C01810=1204.723,228.544,-60.567,-177.311,6.595,148.417
C01811=1204.727,228.295,-60.541,-177.313,6.593,148.418
C01812=1204.732,228.047,-60.516,-177.316,6.591,148.418
C01813=1204.736,227.798,-60.490,-177.318,6.589,148.418
C01814=1204.740,227.549,-60.465,-177.321,6.587,148.418
C01815=1204.745,227.300,-60.440,-177.324,6.586,148.419
C01816=1204.749,227.052,-60.414,-177.326,6.584,148.419
C01817=1204.755,226.803,-60.389,-177.329,6.581,148.419
C01818=1204.759,226.554,-60.364,-177.332,6.579,148.420
C01819=1204.762,226.306,-60.338,-177.334,6.577,148.420
C01820=1204.767,226.057,-60.314,-177.337,6.575,148.420
C01821=1204.772,225.808,-60.288,-177.339,6.573,148.420
C01822=1204.776,225.560,-60.263,-177.342,6.571,148.421
C01823=1204.781,225.311,-60.238,-177.344,6.569,148.421
C01824=1204.786,225.063,-60.212,-177.347,6.567,148.421
C01825=1204.790,224.814,-60.187,-177.350,6.565,148.421
C01826=1204.794,224.565,-60.162,-177.352,6.563,148.422
C01827=1204.799,224.316,-60.137,-177.355,6.561,148.422
C01828=1204.804,224.068,-60.112,-177.358,6.559,148.422
C01829=1204.808,223.819,-60.086,-177.360,6.557,148.423
C01830=1204.813,223.570,-60.062,-177.362,6.555,148.423
C01831=1204.817,223.321,-60.036,-177.365,6.553,148.423
C01832=1204.821,223.072,-60.011,-177.368,6.551,148.423
C01833=1204.826,222.824,-59.986,-177.371,6.549,148.424
C01834=1204.830,222.575,-59.961,-177.373,6.547,148.424
C01835=1204.835,222.327,-59.936,-177.376,6.545,148.424
C01836=1204.840,222.078,-59.912,-177.378,6.543,148.424
C01837=1204.844,221.829,-59.886,-177.381,6.541,148.425
C01838=1204.849,221.581,-59.861,-177.384,6.539,148.425
C01839=1204.853,221.332,-59.835,-177.386,6.537,148.425
C01840=1204.858,221.084,-59.811,-177.388,6.535,148.426
C01841=1204.862,220.834,-59.786,-177.391,6.533,148.426
C01842=1204.867,220.586,-59.761,-177.394,6.531,148.426
C01843=1204.872,220.337,-59.736,-177.397,6.529,148.427
C01844=1204.876,220.089,-59.711,-177.399,6.527,148.427
C01845=1204.880,219.839,-59.686,-177.402,6.525,148.427
C01846=1204.885,219.591,-59.661,-177.404,6.523,148.427
C01847=1204.889,219.342,-59.636,-177.407,6.521,148.428
C01848=1204.894,219.093,-59.612,-177.410,6.519,148.428
C01849=1204.899,218.845,-59.587,-177.412,6.517,148.428
C01850=1204.903,218.596,-59.562,-177.414,6.515,148.428
C01851=1204.908,218.347,-59.537,-177.417,6.514,148.429
C01852=1204.912,218.098,-59.512,-177.420,6.511,148.429
C01853=1204.916,217.850,-59.487,-177.423,6.509,148.429
C01854=1204.921,217.601,-59.462,-177.425,6.507,148.430
C01855=1204.925,217.352,-59.438,-177.428,6.505,148.430
C01856=1204.930,217.104,-59.413,-177.430,6.503,148.430
C01857=1204.935,216.855,-59.388,-177.433,6.501,148.430
C01858=1204.939,216.606,-59.364,-177.436,6.500,148.431
C01859=1204.944,216.357,-59.339,-177.438,6.498,148.431
C01860=1204.948,216.109,-59.314,-177.441,6.496,148.431
C01861=1204.953,215.860,-59.290,-177.443,6.494,148.432
C01862=1204.957,215.611,-59.264,-177.446,6.492,148.432
C01863=1204.962,215.363,-59.240,-177.449,6.489,148.432
C01864=1204.967,215.114,-59.215,-177.451,6.487,148.433
C01865=1204.971,214.865,-59.191,-177.454,6.486,148.433
C01866=1204.976,214.616,-59.166,-177.457,6.484,148.433
C01867=1204.980,214.368,-59.142,-177.459,6.482,148.433
C01868=1204.985,214.118,-59.117,-177.462,6.480,148.434
C01869=1204.989,213.870,-59.093,-177.464,6.478,148.434
C01870=1204.994,213.622,-59.068,-177.467,6.476,148.434
C01871=1204.998,213.373,-59.043,-177.469,6.474,148.435
C01872=1205.003,213.124,-59.019,-177.472,6.472,148.435
C01873=1205.007,212.876,-58.994,-177.475,6.471,148.435
C01874=1205.012,212.626,-58.969,-177.477,6.468,148.435
C01875=1205.016,212.378,-58.945,-177.480,6.467,148.436
C01876=1205.021,212.129,-58.921,-177.482,6.465,148.436
C01877=1205.025,211.880,-58.896,-177.485,6.463,148.436
C01878=1205.030,211.631,-58.872,-177.488,6.460,148.437
C01879=1205.035,211.361,-58.845,-177.491,6.458,148.437
C01880=1205.040,211.090,-58.819,-177.493,6.457,148.437
C01881=1205.045,210.820,-58.792,-177.496,6.455,148.438
C01882=1205.050,210.549,-58.766,-177.499,6.452,148.438
C01883=1205.054,210.301,-58.742,-177.502,6.450,148.438
C01884=1205.059,210.052,-58.717,-177.504,6.448,148.439
C01885=1205.063,209.803,-58.692,-177.507,6.447,148.439
C01886=1205.067,209.555,-58.668,-177.510,6.445,148.439
C01887=1205.073,209.305,-58.644,-177.512,6.443,148.440
C01888=1205.077,209.057,-58.620,-177.515,6.441,148.440
C01889=1205.082,208.808,-58.595,-177.517,6.439,148.440
C01890=1205.086,208.559,-58.571,-177.520,6.437,148.441
C01891=1205.091,208.311,-58.547,-177.523,6.435,148.441
C01892=1205.096,208.062,-58.523,-177.525,6.433,148.441
C01893=1205.100,207.813,-58.498,-177.528,6.432,148.442
C01894=1205.104,207.564,-58.475,-177.530,6.430,148.442
C01895=1205.109,207.315,-58.450,-177.533,6.428,148.442
C01896=1205.114,207.067,-58.426,-177.536,6.426,148.443
C01897=1205.118,206.818,-58.402,-177.538,6.424,148.443
C01898=1205.123,206.569,-58.377,-177.541,6.422,148.443
C01899=1205.127,206.320,-58.354,-177.543,6.420,148.443
C01900=1205.132,206.071,-58.329,-177.546,6.418,148.444
C01901=1205.136,205.823,-58.305,-177.549,6.417,148.444
C01902=1205.142,205.574,-58.281,-177.551,6.415,148.444
C01903=1205.146,205.325,-58.257,-177.554,6.413,148.445
C01904=1205.150,205.076,-58.233,-177.556,6.411,148.445
C01905=1205.154,204.828,-58.209,-177.559,6.409,148.445
C01906=1205.160,204.578,-58.185,-177.562,6.408,148.446
C01907=1205.164,204.330,-58.161,-177.564,6.406,148.446
C01908=1205.168,204.082,-58.137,-177.567,6.404,148.446
C01909=1205.173,203.833,-58.113,-177.569,6.402,148.447
C01910=1205.178,203.583,-58.088,-177.572,6.400,148.447
C01911=1205.182,203.334,-58.065,-177.575,6.398,148.447
C01912=1205.187,203.086,-58.041,-177.577,6.396,148.448
C01913=1205.191,202.837,-58.017,-177.580,6.394,148.448
C01914=1205.196,202.588,-57.993,-177.582,6.393,148.448
C01915=1205.200,202.340,-57.969,-177.585,6.391,148.449
C01916=1205.206,202.091,-57.945,-177.588,6.389,148.449
C01917=1205.209,201.841,-57.921,-177.590,6.387,148.449
C01918=1205.214,201.593,-57.897,-177.593,6.385,148.450
C01919=1205.219,201.344,-57.874,-177.596,6.383,148.450
C01920=1205.223,201.096,-57.849,-177.598,6.382,148.450
C01921=1205.228,200.847,-57.826,-177.601,6.380,148.451
C01922=1205.232,200.598,-57.802,-177.604,6.378,148.451
C01923=1205.237,200.349,-57.778,-177.606,6.376,148.451
C01924=1205.242,200.100,-57.754,-177.608,6.374,148.451
C01925=1205.247,199.851,-57.731,-177.611,6.372,148.452
C01926=1205.251,199.603,-57.707,-177.614,6.370,148.452
C01927=1205.256,199.354,-57.683,-177.616,6.369,148.453
C01928=1205.260,199.105,-57.660,-177.619,6.367,148.453
C01929=1205.264,198.856,-57.635,-177.622,6.365,148.453
C01930=1205.269,198.607,-57.612,-177.624,6.363,148.454
C01931=1205.273,198.358,-57.588,-177.627,6.361,148.454
C01932=1205.278,198.109,-57.565,-177.630,6.359,148.454
C01933=1205.283,197.860,-57.541,-177.632,6.358,148.455
C01934=1205.287,197.612,-57.517,-177.635,6.356,148.455
C01935=1205.292,197.363,-57.494,-177.638,6.354,148.455
C01936=1205.296,197.114,-57.470,-177.640,6.352,148.456
C01937=1205.301,196.865,-57.446,-177.643,6.350,148.456
C01938=1205.306,196.616,-57.423,-177.646,6.349,148.456
C01939=1205.310,196.368,-57.399,-177.648,6.347,148.457
C01940=1205.315,196.119,-57.376,-177.651,6.345,148.457
C01941=1205.319,195.870,-57.352,-177.654,6.343,148.457
C01942=1205.324,195.621,-57.329,-177.656,6.341,148.458
C01943=1205.328,195.372,-57.305,-177.659,6.339,148.458
C01944=1205.333,195.123,-57.281,-177.662,6.338,148.458
C01945=1205.338,194.874,-57.258,-177.664,6.337,148.459
C01946=1205.343,194.625,-57.235,-177.666,6.335,148.459
C01947=1205.347,194.377,-57.211,-177.669,6.333,148.459
C01948=1205.352,194.128,-57.187,-177.672,6.331,148.460
C01949=1205.356,193.879,-57.164,-177.674,6.329,148.460
C01950=1205.361,193.630,-57.141,-177.677,6.327,148.461
C01951=1205.366,193.381,-57.117,-177.680,6.326,148.461
C01952=1205.370,193.132,-57.093,-177.682,6.324,148.461
C01953=1205.374,192.884,-57.070,-177.685,6.322,148.462
C01954=1205.379,192.635,-57.047,-177.687,6.320,148.462
C01955=1205.384,192.386,-57.024,-177.690,6.318,148.462
C01956=1205.389,192.137,-57.001,-177.693,6.317,148.463
C01957=1205.393,191.888,-56.977,-177.695,6.315,148.463
C01958=1205.398,191.639,-56.954,-177.698,6.313,148.463
C01959=1205.403,191.391,-56.930,-177.700,6.312,148.464
C01960=1205.407,191.142,-56.907,-177.703,6.310,148.464
C01961=1205.411,190.893,-56.884,-177.705,6.308,148.464
C01962=1205.416,190.644,-56.860,-177.708,6.306,148.465
C01963=1205.421,190.395,-56.837,-177.711,6.305,148.465
C01964=1205.425,190.146,-56.814,-177.713,6.303,148.465
C01965=1205.430,189.897,-56.790,-177.716,6.301,148.466
C01966=1205.435,189.649,-56.768,-177.719,6.299,148.466
C01967=1205.439,189.400,-56.745,-177.721,6.297,148.466
C01968=1205.444,189.151,-56.721,-177.724,6.296,148.467
C01969=1205.449,188.902,-56.698,-177.727,6.294,148.467
C01970=1205.453,188.653,-56.674,-177.729,6.293,148.468
C01971=1205.457,188.404,-56.652,-177.731,6.291,148.468
C01972=1205.462,188.155,-56.628,-177.734,6.289,148.468
C01973=1205.467,187.906,-56.605,-177.737,6.287,148.469
C01974=1205.472,187.658,-56.582,-177.739,6.286,148.469
C01975=1205.476,187.409,-56.559,-177.742,6.284,148.469
C01976=1205.481,187.160,-56.536,-177.745,6.282,148.470
C01977=1205.486,186.910,-56.513,-177.747,6.280,148.470
C01978=1205.490,186.661,-56.490,-177.750,6.278,148.470
C01979=1205.494,186.412,-56.467,-177.752,6.277,148.471
C01980=1205.500,186.164,-56.444,-177.755,6.275,148.471
C01981=1205.504,185.915,-56.421,-177.757,6.274,148.471
C01982=1205.508,185.666,-56.398,-177.760,6.272,148.472
C01983=1205.514,185.397,-56.373,-177.763,6.270,148.472
C01984=1205.519,185.127,-56.348,-177.766,6.269,148.473
C01985=1205.524,184.857,-56.324,-177.769,6.267,148.473
C01986=1205.529,184.588,-56.298,-177.772,6.264,148.473
C01987=1205.533,184.339,-56.276,-177.774,6.263,148.474
C01988=1205.538,184.090,-56.252,-177.777,6.261,148.474
C01989=1205.543,183.842,-56.229,-177.779,6.259,148.475
C01990=1205.547,183.592,-56.207,-177.782,6.258,148.475
C01991=1205.552,183.343,-56.184,-177.785,6.256,148.475
C01992=1205.556,183.094,-56.161,-177.787,6.254,148.476
C01993=1205.561,182.845,-56.139,-177.790,6.253,148.476
C01994=1205.566,182.596,-56.116,-177.793,6.251,148.476
C01995=1205.570,182.348,-56.093,-177.795,6.250,148.477
C01996=1205.575,182.099,-56.069,-177.798,6.248,148.477
C01997=1205.579,181.849,-56.047,-177.800,6.246,148.478
C01998=1205.584,181.601,-56.024,-177.803,6.244,148.478
C01999=1205.588,181.352,-56.002,-177.806,6.242,148.478
C02000=1205.593,181.103,-55.979,-177.808,6.241,148.479
C02001=1205.598,180.854,-55.956,-177.810,6.240,148.479
C02002=1205.603,180.606,-55.933,-177.813,6.238,148.479
C02003=1205.608,180.356,-55.911,-177.816,6.236,148.480
C02004=1205.612,180.107,-55.888,-177.818,6.234,148.480
C02005=1205.617,179.858,-55.866,-177.821,6.232,148.480
C02006=1205.621,179.610,-55.843,-177.824,6.231,148.481
C02007=1205.626,179.361,-55.819,-177.827,6.229,148.481
C02008=1205.630,179.111,-55.797,-177.829,6.228,148.482
C02009=1205.635,178.863,-55.774,-177.832,6.226,148.482
C02010=1205.640,178.613,-55.752,-177.834,6.225,148.483
C02011=1205.644,178.364,-55.729,-177.837,6.223,148.483
C02012=1205.649,178.116,-55.707,-177.840,6.221,148.483
C02013=1205.653,177.867,-55.685,-177.842,6.219,148.484
C02014=1205.658,177.617,-55.662,-177.844,6.218,148.484
C02015=1205.663,177.369,-55.639,-177.847,6.216,148.484
C02016=1205.668,177.120,-55.617,-177.850,6.215,148.485
C02017=1205.672,176.871,-55.594,-177.853,6.213,148.485
C02018=1205.677,176.622,-55.572,-177.856,6.211,148.486
C02019=1205.681,176.373,-55.549,-177.858,6.210,148.486
C02020=1205.686,176.124,-55.527,-177.860,6.208,148.486
C02021=1205.691,175.876,-55.504,-177.863,6.207,148.487
C02022=1205.695,175.626,-55.482,-177.866,6.205,148.487
C02023=1205.700,175.377,-55.459,-177.868,6.203,148.487
C02024=1205.705,175.129,-55.437,-177.871,6.201,148.488
C02025=1205.709,174.879,-55.415,-177.873,6.200,148.488
C02026=1205.714,174.631,-55.392,-177.876,6.198,148.489
C02027=1205.718,174.382,-55.370,-177.879,6.197,148.489
C02028=1205.723,174.132,-55.348,-177.882,6.195,148.489
C02029=1205.728,173.884,-55.325,-177.884,6.193,148.490
C02030=1205.732,173.635,-55.303,-177.886,6.192,148.490
C02031=1205.737,173.386,-55.281,-177.889,6.191,148.491
C02032=1205.742,173.137,-55.258,-177.892,6.189,148.491
C02033=1205.746,172.888,-55.236,-177.894,6.187,148.491
C02034=1205.751,172.639,-55.214,-177.897,6.185,148.492
C02035=1205.756,172.390,-55.191,-177.900,6.185,148.492
C02036=1205.761,172.141,-55.169,-177.902,6.183,148.493
C02037=1205.765,171.892,-55.147,-177.905,6.181,148.493
C02038=1205.770,171.643,-55.125,-177.908,6.179,148.493
C02039=1205.774,171.394,-55.102,-177.910,6.177,148.494
C02040=1205.779,171.145,-55.080,-177.912,6.176,148.494
C02041=1205.784,170.896,-55.058,-177.915,6.174,148.494
C02042=1205.789,170.647,-55.035,-177.918,6.173,148.495
C02043=1205.793,170.398,-55.014,-177.921,6.171,148.495
C02044=1205.797,170.149,-54.991,-177.923,6.170,148.496
C02045=1205.802,169.901,-54.969,-177.926,6.168,148.496
C02046=1205.807,169.651,-54.947,-177.928,6.167,148.497
C02047=1205.812,169.402,-54.925,-177.931,6.165,148.497
C02048=1205.816,169.153,-54.903,-177.934,6.163,148.497
C02049=1205.821,168.904,-54.881,-177.936,6.162,148.498
C02050=1205.825,168.656,-54.858,-177.939,6.161,148.498
C02051=1205.831,168.407,-54.836,-177.941,6.159,148.499
C02052=1205.835,168.157,-54.814,-177.944,6.157,148.499
C02053=1205.840,167.909,-54.792,-177.946,6.156,148.499
C02054=1205.844,167.659,-54.770,-177.949,6.154,148.500
C02055=1205.849,167.411,-54.749,-177.952,6.153,148.500
C02056=1205.853,167.161,-54.727,-177.955,6.151,148.501
C02057=1205.859,166.912,-54.704,-177.957,6.150,148.501
C02058=1205.863,166.663,-54.682,-177.959,6.148,148.501
C02059=1205.868,166.415,-54.661,-177.962,6.146,148.502
C02060=1205.872,166.165,-54.639,-177.965,6.145,148.502
C02061=1205.877,165.917,-54.617,-177.967,6.144,148.503
C02062=1205.882,165.667,-54.595,-177.970,6.142,148.503
C02063=1205.886,165.419,-54.573,-177.973,6.140,148.504
C02064=1205.891,165.169,-54.551,-177.975,6.138,148.504
C02065=1205.896,164.921,-54.530,-177.978,6.138,148.504
C02066=1205.901,164.672,-54.507,-177.980,6.136,148.505
C02067=1205.905,164.422,-54.485,-177.983,6.134,148.505
C02068=1205.910,164.174,-54.463,-177.986,6.132,148.506
C02069=1205.915,163.924,-54.441,-177.988,6.131,148.506
C02070=1205.919,163.676,-54.420,-177.991,6.130,148.506
C02071=1205.924,163.426,-54.398,-177.993,6.128,148.507
C02072=1205.929,163.178,-54.376,-177.997,6.126,148.507
C02073=1205.933,162.929,-54.354,-177.999,6.125,148.508
C02074=1205.938,162.679,-54.333,-178.001,6.124,148.508
C02075=1205.943,162.430,-54.311,-178.004,6.122,148.508
C02076=1205.947,162.181,-54.289,-178.006,6.121,148.509
C02077=1205.952,161.932,-54.268,-178.009,6.119,148.509
C02078=1205.957,161.684,-54.246,-178.012,6.118,148.510
C02079=1205.961,161.434,-54.224,-178.015,6.116,148.510
C02080=1205.966,161.185,-54.203,-178.017,6.115,148.511
C02081=1205.971,160.936,-54.181,-178.019,6.113,148.511
C02082=1205.975,160.687,-54.159,-178.023,6.112,148.512
C02083=1205.980,160.439,-54.137,-178.025,6.111,148.512
C02084=1205.985,160.189,-54.115,-178.027,6.109,148.512
C02085=1205.990,159.940,-54.094,-178.030,6.107,148.513
C02086=1205.995,159.691,-54.073,-178.033,6.105,148.513
C02087=1205.999,159.422,-54.050,-178.036,6.104,148.514
C02088=1206.005,159.154,-54.026,-178.038,6.103,148.514
C02089=1206.009,158.885,-54.003,-178.041,6.101,148.515
C02090=1206.015,158.615,-53.980,-178.044,6.100,148.515
C02091=1206.019,158.366,-53.958,-178.046,6.098,148.515
C02092=1206.024,158.117,-53.936,-178.049,6.096,148.516
C02093=1206.029,157.868,-53.915,-178.052,6.095,148.516
C02094=1206.033,157.619,-53.894,-178.054,6.094,148.517
C02095=1206.038,157.370,-53.872,-178.057,6.092,148.517
C02096=1206.043,157.121,-53.851,-178.059,6.091,148.517
C02097=1206.048,156.872,-53.829,-178.062,6.089,148.518
C02098=1206.052,156.623,-53.807,-178.065,6.087,148.518
C02099=1206.057,156.374,-53.786,-178.068,6.086,148.519
C02100=1206.062,156.125,-53.765,-178.070,6.085,148.519
C02101=1206.066,155.875,-53.744,-178.073,6.083,148.520
C02102=1206.071,155.627,-53.722,-178.076,6.081,148.520
C02103=1206.075,155.378,-53.701,-178.078,6.080,148.521
C02104=1206.081,155.129,-53.680,-178.080,6.079,148.521
C02105=1206.085,154.880,-53.658,-178.083,6.077,148.521
C02106=1206.089,154.631,-53.637,-178.086,6.076,148.522
C02107=1206.094,154.382,-53.615,-178.088,6.074,148.522
C02108=1206.099,154.133,-53.595,-178.091,6.073,148.523
C02109=1206.104,153.883,-53.572,-178.093,6.072,148.523
C02110=1206.109,153.634,-53.552,-178.096,6.070,148.524
C02111=1206.113,153.386,-53.530,-178.099,6.068,148.524
C02112=1206.118,153.137,-53.509,-178.101,6.068,148.524
C02113=1206.122,152.887,-53.487,-178.104,6.066,148.525
C02114=1206.128,152.638,-53.466,-178.107,6.064,148.525
C02115=1206.132,152.390,-53.445,-178.109,6.063,148.526
C02116=1206.137,152.140,-53.424,-178.112,6.061,148.526
C02117=1206.141,151.891,-53.402,-178.115,6.060,148.527
C02118=1206.146,151.642,-53.381,-178.117,6.059,148.527
C02119=1206.151,151.393,-53.361,-178.120,6.057,148.528
C02120=1206.156,151.144,-53.339,-178.122,6.055,148.528
C02121=1206.161,150.895,-53.318,-178.125,6.055,148.529
C02122=1206.164,150.646,-53.297,-178.128,6.053,148.529
C02123=1206.170,150.397,-53.276,-178.130,6.051,148.529
C02124=1206.175,150.147,-53.255,-178.132,6.050,148.530
C02125=1206.179,149.899,-53.234,-178.135,6.049,148.530
C02126=1206.184,149.650,-53.213,-178.138,6.048,148.531
C02127=1206.189,149.400,-53.192,-178.140,6.046,148.531
C02128=1206.193,149.151,-53.170,-178.143,6.044,148.531
C02129=1206.198,148.902,-53.150,-178.146,6.044,148.532
C02130=1206.203,148.653,-53.129,-178.148,6.042,148.532
C02131=1206.207,148.405,-53.107,-178.151,6.040,148.533
C02132=1206.212,148.155,-53.086,-178.153,6.039,148.533
C02133=1206.217,147.906,-53.066,-178.156,6.038,148.534
C02134=1206.221,147.656,-53.045,-178.159,6.036,148.534
C02135=1206.226,147.408,-53.023,-178.161,6.035,148.535
C02136=1206.231,147.159,-53.003,-178.164,6.033,148.535
C02137=1206.236,146.910,-52.982,-178.166,6.033,148.536
C02138=1206.240,146.661,-52.961,-178.169,6.031,148.536
C02139=1206.245,146.412,-52.940,-178.172,6.029,148.537
C02140=1206.250,146.163,-52.919,-178.174,6.028,148.537
C02141=1206.255,145.914,-52.898,-178.177,6.027,148.537
C02142=1206.260,145.665,-52.877,-178.180,6.025,148.538
C02143=1206.264,145.415,-52.857,-178.182,6.024,148.538
C02144=1206.269,145.166,-52.836,-178.185,6.022,148.539
C02145=1206.273,144.917,-52.815,-178.187,6.021,148.539
C02146=1206.278,144.668,-52.794,-178.190,6.020,148.540
C02147=1206.283,144.419,-52.773,-178.193,6.018,148.540
C02148=1206.288,144.170,-52.752,-178.195,6.017,148.541
C02149=1206.292,143.921,-52.732,-178.198,6.016,148.541
C02150=1206.297,143.672,-52.711,-178.200,6.015,148.542
C02151=1206.302,143.423,-52.691,-178.203,6.013,148.542
C02152=1206.307,143.173,-52.670,-178.206,6.012,148.543
C02153=1206.312,142.924,-52.649,-178.208,6.011,148.543
C02154=1206.317,142.675,-52.628,-178.211,6.009,148.543
C02155=1206.320,142.426,-52.607,-178.213,6.008,148.544
C02156=1206.325,142.177,-52.586,-178.216,6.006,148.544
C02157=1206.330,141.928,-52.566,-178.219,6.005,148.545
C02158=1206.334,141.679,-52.545,-178.221,6.004,148.545
C02159=1206.339,141.430,-52.524,-178.224,6.002,148.546
C02160=1206.344,141.181,-52.504,-178.226,6.001,148.546
C02161=1206.349,140.932,-52.483,-178.229,6.000,148.547
C02162=1206.354,140.683,-52.462,-178.232,5.998,148.547
C02163=1206.359,140.433,-52.441,-178.234,5.997,148.548
C02164=1206.363,140.184,-52.422,-178.237,5.996,148.548
C02165=1206.368,139.935,-52.401,-178.239,5.995,148.549
C02166=1206.373,139.686,-52.380,-178.242,5.993,148.549
C02167=1206.377,139.437,-52.360,-178.245,5.992,148.550
C02168=1206.383,139.187,-52.339,-178.247,5.990,148.550
C02169=1206.387,138.938,-52.319,-178.250,5.989,148.550
C02170=1206.392,138.689,-52.298,-178.253,5.988,148.551
C02171=1206.397,138.440,-52.277,-178.255,5.986,148.551
C02172=1206.401,138.191,-52.257,-178.257,5.985,148.552
C02173=1206.406,137.942,-52.237,-178.261,5.984,148.552
C02174=1206.411,137.693,-52.216,-178.263,5.982,148.553
C02175=1206.415,137.443,-52.196,-178.265,5.981,148.553
C02176=1206.420,137.195,-52.176,-178.269,5.980,148.554
C02177=1206.425,136.945,-52.155,-178.271,5.979,148.554
C02178=1206.430,136.697,-52.135,-178.273,5.977,148.555
C02179=1206.435,136.448,-52.114,-178.276,5.976,148.555
C02180=1206.439,136.198,-52.095,-178.279,5.975,148.556
C02181=1206.444,135.949,-52.074,-178.281,5.974,148.556
C02182=1206.449,135.700,-52.053,-178.284,5.972,148.557
C02183=1206.453,135.451,-52.033,-178.287,5.970,148.557
C02184=1206.459,135.202,-52.012,-178.289,5.969,148.557
C02185=1206.463,134.953,-51.992,-178.292,5.968,148.558
C02186=1206.468,134.704,-51.972,-178.294,5.967,148.558
C02187=1206.472,134.455,-51.952,-178.297,5.966,148.559
C02188=1206.478,134.205,-51.931,-178.299,5.965,148.559
C02189=1206.482,133.956,-51.911,-178.302,5.963,148.560
C02190=1206.487,133.707,-51.891,-178.305,5.962,148.560
C02191=1206.492,133.438,-51.869,-178.307,5.960,148.561
C02192=1206.497,133.170,-51.847,-178.310,5.959,148.561
C02193=1206.502,132.901,-51.825,-178.313,5.957,148.562
C02194=1206.507,132.633,-51.804,-178.316,5.957,148.562
C02195=1206.513,132.383,-51.783,-178.318,5.955,148.563
C02196=1206.517,132.134,-51.763,-178.321,5.954,148.563
C02197=1206.521,131.885,-51.743,-178.324,5.952,148.564
C02198=1206.527,131.636,-51.723,-178.326,5.951,148.564
C02199=1206.531,131.387,-51.703,-178.329,5.950,148.565
C02200=1206.536,131.138,-51.683,-178.332,5.948,148.565
C02201=1206.541,130.888,-51.662,-178.334,5.948,148.566
C02202=1206.546,130.639,-51.642,-178.337,5.946,148.566
C02203=1206.550,130.390,-51.622,-178.339,5.945,148.567
C02204=1206.555,130.141,-51.602,-178.342,5.943,148.567
C02205=1206.560,129.892,-51.583,-178.344,5.943,148.568
C02206=1206.564,129.643,-51.562,-178.348,5.941,148.568
C02207=1206.569,129.394,-51.543,-178.350,5.940,148.569
C02208=1206.574,129.145,-51.522,-178.352,5.938,148.569
C02209=1206.578,128.895,-51.503,-178.355,5.938,148.570
C02210=1206.584,128.646,-51.482,-178.358,5.936,148.570
C02211=1206.589,128.397,-51.462,-178.360,5.935,148.571
C02212=1206.593,128.148,-51.442,-178.363,5.934,148.571
C02213=1206.598,127.898,-51.422,-178.365,5.933,148.572
C02214=1206.603,127.649,-51.402,-178.368,5.931,148.572
C02215=1206.608,127.401,-51.383,-178.370,5.930,148.573
C02216=1206.612,127.152,-51.362,-178.373,5.929,148.573
C02217=1206.617,126.902,-51.343,-178.376,5.928,148.574
C02218=1206.622,126.653,-51.322,-178.378,5.926,148.574
C02219=1206.626,126.404,-51.303,-178.381,5.925,148.575
C02220=1206.632,126.155,-51.283,-178.384,5.924,148.575
C02221=1206.636,125.906,-51.263,-178.386,5.923,148.576
C02222=1206.641,125.656,-51.243,-178.389,5.921,148.576
C02223=1206.646,125.407,-51.224,-178.391,5.920,148.576
C02224=1206.651,125.158,-51.204,-178.394,5.919,148.577
C02225=1206.655,124.909,-51.184,-178.396,5.918,148.577
C02226=1206.660,124.660,-51.164,-178.399,5.917,148.578
C02227=1206.664,124.410,-51.144,-178.402,5.916,148.578
C02228=1206.670,124.161,-51.125,-178.405,5.914,148.579
C02229=1206.674,123.912,-51.104,-178.407,5.913,148.579
C02230=1206.679,123.663,-51.085,-178.410,5.911,148.580
C02231=1206.684,123.413,-51.065,-178.412,5.911,148.581
C02232=1206.689,123.164,-51.046,-178.415,5.909,148.581
C02233=1206.694,122.916,-51.025,-178.417,5.908,148.582
C02234=1206.698,122.666,-51.006,-178.420,5.908,148.582
C02235=1206.703,122.417,-50.987,-178.423,5.906,148.583
C02236=1206.708,122.168,-50.967,-178.425,5.905,148.583
C02237=1206.712,121.919,-50.947,-178.428,5.903,148.583
C02238=1206.717,121.669,-50.927,-178.430,5.903,148.584
C02239=1206.722,121.420,-50.908,-178.433,5.901,148.584
C02240=1206.727,121.171,-50.888,-178.435,5.900,148.585
C02241=1206.731,120.922,-50.868,-178.438,5.899,148.585
C02242=1206.737,120.673,-50.849,-178.441,5.898,148.586
C02243=1206.741,120.423,-50.829,-178.443,5.896,148.586
C02244=1206.745,120.174,-50.810,-178.446,5.896,148.587
C02245=1206.751,119.925,-50.791,-178.449,5.894,148.587
C02246=1206.756,119.676,-50.771,-178.451,5.893,148.588
C02247=1206.760,119.427,-50.751,-178.454,5.892,148.589
C02248=1206.765,119.178,-50.731,-178.456,5.891,148.589
C02249=1206.770,118.928,-50.712,-178.459,5.890,148.590
C02250=1206.775,118.680,-50.693,-178.461,5.888,148.590
C02251=1206.779,118.430,-50.673,-178.464,5.888,148.591
C02252=1206.784,118.181,-50.654,-178.467,5.886,148.591
C02253=1206.789,117.932,-50.634,-178.469,5.885,148.592
C02254=1206.794,117.682,-50.615,-178.472,5.883,148.592
C02255=1206.798,117.433,-50.596,-178.475,5.883,148.593
C02256=1206.804,117.184,-50.576,-178.477,5.881,148.593
C02257=1206.808,116.935,-50.557,-178.480,5.880,148.594
C02258=1206.814,116.686,-50.537,-178.482,5.880,148.594
C02259=1206.818,116.436,-50.518,-178.485,5.878,148.595
C02260=1206.822,116.187,-50.499,-178.487,5.877,148.595
C02261=1206.828,115.938,-50.479,-178.490,5.875,148.596
C02262=1206.832,115.688,-50.460,-178.493,5.875,148.596
C02263=1206.838,115.440,-50.440,-178.495,5.873,148.597
C02264=1206.842,115.190,-50.421,-178.498,5.872,148.597
C02265=1206.847,114.941,-50.402,-178.500,5.871,148.598
C02266=1206.852,114.692,-50.382,-178.503,5.870,148.598
C02267=1206.856,114.443,-50.363,-178.505,5.869,148.599
C02268=1206.861,114.194,-50.344,-178.509,5.868,148.599
C02269=1206.866,113.944,-50.324,-178.511,5.867,148.600
C02270=1206.871,113.695,-50.305,-178.514,5.865,148.600
C02271=1206.875,113.446,-50.286,-178.516,5.864,148.601
C02272=1206.881,113.197,-50.267,-178.519,5.864,148.601
C02273=1206.885,112.948,-50.247,-178.521,5.862,148.602
C02274=1206.889,112.698,-50.228,-178.524,5.861,148.602
C02275=1206.895,112.449,-50.210,-178.527,5.860,148.603
C02276=1206.900,112.199,-50.190,-178.529,5.859,148.603
C02277=1206.904,111.951,-50.171,-178.531,5.858,148.604
C02278=1206.909,111.701,-50.152,-178.535,5.857,148.605
C02279=1206.914,111.453,-50.133,-178.537,5.856,148.605
C02280=1206.919,111.203,-50.113,-178.540,5.854,148.606
C02281=1206.924,110.954,-50.095,-178.542,5.853,148.606
C02282=1206.928,110.704,-50.076,-178.545,5.853,148.607
C02283=1206.934,110.455,-50.056,-178.547,5.851,148.607
C02284=1206.938,110.206,-50.037,-178.550,5.850,148.608
C02285=1206.943,109.957,-50.018,-178.553,5.849,148.608
C02286=1206.948,109.707,-49.999,-178.555,5.848,148.609
C02287=1206.953,109.459,-49.980,-178.557,5.847,148.609
C02288=1206.957,109.209,-49.961,-178.561,5.846,148.610
C02289=1206.962,108.960,-49.942,-178.563,5.845,148.610
C02290=1206.967,108.710,-49.923,-178.566,5.843,148.611
C02291=1206.972,108.461,-49.904,-178.568,5.842,148.611
C02292=1206.976,108.212,-49.885,-178.571,5.842,148.612
C02293=1206.982,107.963,-49.865,-178.573,5.840,148.612
C02294=1206.987,107.714,-49.847,-178.576,5.840,148.613
C02295=1206.991,107.445,-49.826,-178.579,5.838,148.613
C02296=1206.997,107.177,-49.806,-178.581,5.837,148.614
C02297=1207.001,106.909,-49.786,-178.584,5.836,148.615
C02298=1207.007,106.640,-49.766,-178.587,5.835,148.615
C02299=1207.011,106.391,-49.747,-178.590,5.833,148.616
C02300=1207.017,106.142,-49.727,-178.592,5.833,148.616
C02301=1207.022,105.893,-49.709,-178.595,5.831,148.617
C02302=1207.026,105.643,-49.690,-178.598,5.830,148.617
C02303=1207.031,105.395,-49.671,-178.600,5.830,148.618
C02304=1207.036,105.144,-49.652,-178.603,5.828,148.618
C02305=1207.041,104.896,-49.633,-178.605,5.827,148.619
C02306=1207.046,104.646,-49.615,-178.608,5.827,148.619
C02307=1207.050,104.397,-49.596,-178.610,5.825,148.620
C02308=1207.056,104.148,-49.577,-178.613,5.824,148.620
C02309=1207.060,103.898,-49.558,-178.615,5.823,148.621
C02310=1207.066,103.649,-49.540,-178.618,5.822,148.622
C02311=1207.070,103.400,-49.521,-178.620,5.821,148.622
C02312=1207.074,103.150,-49.503,-178.624,5.820,148.623
C02313=1207.080,102.902,-49.483,-178.626,5.819,148.623
C02314=1207.084,102.652,-49.465,-178.628,5.818,148.624
C02315=1207.089,102.403,-49.446,-178.632,5.817,148.624
C02316=1207.094,102.154,-49.428,-178.634,5.816,148.625
C02317=1207.098,101.904,-49.409,-178.636,5.815,148.625
C02318=1207.104,101.655,-49.390,-178.639,5.813,148.626
C02319=1207.109,101.406,-49.371,-178.642,5.813,148.626
C02320=1207.113,101.156,-49.353,-178.644,5.812,148.627
C02321=1207.118,100.908,-49.334,-178.647,5.810,148.627
C02322=1207.123,100.658,-49.316,-178.649,5.809,148.628
C02323=1207.127,100.409,-49.297,-178.652,5.809,148.629
C02324=1207.133,100.160,-49.278,-178.655,5.807,148.629
C02325=1207.138,99.911,-49.260,-178.657,5.806,148.630
C02326=1207.142,99.661,-49.241,-178.660,5.806,148.630
C02327=1207.147,99.412,-49.222,-178.662,5.804,148.631
C02328=1207.152,99.163,-49.204,-178.665,5.804,148.631
C02329=1207.156,98.913,-49.185,-178.667,5.803,148.632
C02330=1207.162,98.664,-49.167,-178.670,5.801,148.632
C02331=1207.167,98.415,-49.148,-178.672,5.800,148.633
C02332=1207.171,98.165,-49.130,-178.675,5.800,148.633
C02333=1207.176,97.916,-49.112,-178.678,5.798,148.634
C02334=1207.181,97.667,-49.093,-178.680,5.797,148.634
C02335=1207.186,97.418,-49.075,-178.683,5.797,148.635
C02336=1207.190,97.168,-49.056,-178.686,5.795,148.635
C02337=1207.196,96.919,-49.038,-178.688,5.794,148.636
C02338=1207.201,96.670,-49.019,-178.690,5.794,148.637
C02339=1207.205,96.420,-49.001,-178.694,5.792,148.637
C02340=1207.210,96.171,-48.983,-178.696,5.792,148.638
C02341=1207.215,95.922,-48.965,-178.698,5.791,148.638
C02342=1207.220,95.673,-48.945,-178.702,5.789,148.639
C02343=1207.224,95.423,-48.927,-178.704,5.788,148.639
C02344=1207.229,95.174,-48.909,-178.706,5.788,148.640
C02345=1207.234,94.925,-48.891,-178.708,5.787,148.640
C02346=1207.240,94.675,-48.872,-178.712,5.785,148.641
C02347=1207.244,94.426,-48.853,-178.714,5.785,148.642
C02348=1207.249,94.177,-48.835,-178.716,5.784,148.642
C02349=1207.254,93.928,-48.817,-178.720,5.782,148.643
C02350=1207.259,93.679,-48.799,-178.722,5.781,148.643
C02351=1207.264,93.429,-48.781,-178.724,5.781,148.644
C02352=1207.269,93.179,-48.763,-178.727,5.779,148.644
C02353=1207.273,92.931,-48.744,-178.730,5.779,148.645
C02354=1207.278,92.682,-48.726,-178.732,5.778,148.646
C02355=1207.283,92.432,-48.708,-178.734,5.777,148.646
C02356=1207.288,92.183,-48.690,-178.738,5.776,148.647
C02357=1207.292,91.933,-48.672,-178.740,5.775,148.647
C02358=1207.297,91.684,-48.654,-178.742,5.774,148.648
C02359=1207.302,91.435,-48.636,-178.746,5.773,148.648
C02360=1207.308,91.186,-48.617,-178.748,5.772,148.649
C02361=1207.313,90.936,-48.599,-178.750,5.771,148.649
C02362=1207.317,90.686,-48.581,-178.752,5.770,148.650
C02363=1207.322,90.437,-48.563,-178.756,5.769,148.650
C02364=1207.327,90.188,-48.545,-178.758,5.768,148.651
C02365=1207.331,89.940,-48.526,-178.760,5.767,148.652
C02366=1207.336,89.690,-48.508,-178.764,5.766,148.652
C02367=1207.341,89.441,-48.490,-178.766,5.765,148.653
C02368=1207.345,89.191,-48.472,-178.768,5.765,148.653
C02369=1207.350,88.942,-48.454,-178.771,5.764,148.654
C02370=1207.356,88.692,-48.436,-178.774,5.762,148.654
C02371=1207.361,88.443,-48.419,-178.776,5.762,148.655
C02372=1207.365,88.194,-48.401,-178.778,5.761,148.655
C02373=1207.370,87.945,-48.383,-178.781,5.760,148.656
C02374=1207.375,87.696,-48.365,-178.784,5.759,148.657
C02375=1207.380,87.446,-48.347,-178.786,5.758,148.657
C02376=1207.384,87.197,-48.328,-178.789,5.757,148.658
C02377=1207.389,86.947,-48.310,-178.792,5.756,148.658
C02378=1207.394,86.698,-48.292,-178.794,5.755,148.659
C02379=1207.399,86.449,-48.274,-178.797,5.754,148.659
C02380=1207.404,86.200,-48.256,-178.799,5.753,148.660
C02381=1207.409,85.951,-48.238,-178.802,5.752,148.661
C02382=1207.414,85.702,-48.220,-178.805,5.751,148.661
C02383=1207.419,85.452,-48.203,-178.807,5.750,148.662
C02384=1207.424,85.203,-48.185,-178.810,5.750,148.662
C02385=1207.429,84.953,-48.167,-178.813,5.749,148.663
C02386=1207.433,84.704,-48.149,-178.815,5.748,148.663
C02387=1207.438,84.454,-48.131,-178.818,5.747,148.664
C02388=1207.443,84.205,-48.113,-178.820,5.746,148.664
C02389=1207.448,83.955,-48.096,-178.823,5.745,148.665
C02390=1207.453,83.706,-48.078,-178.826,5.744,148.666
C02391=1207.458,83.457,-48.060,-178.828,5.743,148.666
C02392=1207.462,83.208,-48.042,-178.830,5.743,148.667
C02393=1207.468,82.958,-48.025,-178.834,5.741,148.667
C02394=1207.472,82.709,-48.007,-178.836,5.740,148.668
C02395=1207.477,82.460,-47.989,-178.838,5.740,148.669
C02396=1207.482,82.211,-47.971,-178.840,5.739,148.669
C02397=1207.488,81.961,-47.954,-178.843,5.738,148.670
C02398=1207.492,81.712,-47.936,-178.846,5.737,148.670
C02399=1207.498,81.444,-47.916,-178.849,5.736,148.671
C02400=1207.503,81.175,-47.898,-178.852,5.735,148.671
C02401=1207.508,80.906,-47.878,-178.854,5.734,148.672
C02402=1207.513,80.638,-47.859,-178.857,5.733,148.673
C02403=1207.518,80.389,-47.842,-178.860,5.732,148.673
C02404=1207.522,80.140,-47.824,-178.862,5.731,148.674
C02405=1207.527,79.890,-47.806,-178.865,5.731,148.674
C02406=1207.533,79.641,-47.789,-178.867,5.730,148.675
C02407=1207.537,79.391,-47.771,-178.870,5.729,148.675
C02408=1207.542,79.142,-47.754,-178.873,5.728,148.676
C02409=1207.547,78.893,-47.737,-178.875,5.727,148.677
C02410=1207.552,78.644,-47.719,-178.878,5.726,148.677
C02411=1207.558,78.394,-47.701,-178.880,5.726,148.678
C02412=1207.563,78.145,-47.683,-178.883,5.724,148.679
C02413=1207.567,77.896,-47.667,-178.885,5.723,148.679
C02414=1207.572,77.647,-47.649,-178.888,5.723,148.680
C02415=1207.577,77.397,-47.631,-178.891,5.722,148.680
C02416=1207.582,77.148,-47.614,-178.893,5.721,148.681
C02417=1207.586,76.899,-47.596,-178.896,5.720,148.681
C02418=1207.591,76.649,-47.579,-178.899,5.719,148.682
C02419=1207.596,76.400,-47.561,-178.901,5.718,148.682
C02420=1207.602,76.150,-47.544,-178.903,5.718,148.683
C02421=1207.606,75.901,-47.526,-178.906,5.717,148.684
C02422=1207.611,75.651,-47.509,-178.909,5.715,148.684
C02423=1207.616,75.402,-47.491,-178.911,5.715,148.685
C02424=1207.620,75.153,-47.474,-178.914,5.714,148.685
C02425=1207.625,74.904,-47.456,-178.916,5.713,148.686
C02426=1207.630,74.654,-47.439,-178.919,5.713,148.687
C02427=1207.635,74.406,-47.422,-178.922,5.711,148.687
C02428=1207.640,74.156,-47.405,-178.924,5.711,148.688
C02429=1207.645,73.907,-47.387,-178.927,5.710,148.688
C02430=1207.650,73.657,-47.370,-178.929,5.709,148.689
C02431=1207.655,73.407,-47.353,-178.932,5.708,148.689
C02432=1207.660,73.158,-47.335,-178.934,5.708,148.690
C02433=1207.664,72.909,-47.318,-178.937,5.707,148.691
C02434=1207.669,72.660,-47.300,-178.940,5.706,148.691
C02435=1207.675,72.410,-47.283,-178.942,5.705,148.692
C02436=1207.680,72.161,-47.267,-178.945,5.705,148.692
C02437=1207.685,71.912,-47.249,-178.947,5.704,148.693
C02438=1207.689,71.662,-47.232,-178.950,5.702,148.694
C02439=1207.694,71.412,-47.215,-178.953,5.702,148.694
C02440=1207.699,71.163,-47.197,-178.955,5.701,148.695
C02441=1207.704,70.914,-47.180,-178.958,5.700,148.695
C02442=1207.709,70.664,-47.163,-178.960,5.700,148.696
C02443=1207.714,70.416,-47.146,-178.962,5.699,148.696
C02444=1207.719,70.166,-47.129,-178.965,5.697,148.697
C02445=1207.724,69.916,-47.111,-178.968,5.697,148.698
C02446=1207.728,69.667,-47.094,-178.971,5.696,148.698
C02447=1207.734,69.418,-47.077,-178.973,5.695,148.699
C02448=1207.738,69.168,-47.060,-178.976,5.695,148.699
C02449=1207.744,68.919,-47.043,-178.978,5.694,148.700
C02450=1207.748,68.670,-47.026,-178.981,5.692,148.701
C02451=1207.753,68.420,-47.009,-178.983,5.692,148.701
C02452=1207.758,68.171,-46.992,-178.986,5.691,148.702
C02453=1207.763,67.921,-46.975,-178.988,5.690,148.702
C02454=1207.767,67.672,-46.957,-178.991,5.690,148.703
C02455=1207.773,67.423,-46.940,-178.994,5.689,148.704
C02456=1207.777,67.174,-46.924,-178.997,5.688,148.704
C02457=1207.783,66.924,-46.906,-178.999,5.687,148.705
C02458=1207.787,66.674,-46.890,-179.002,5.686,148.705
C02459=1207.793,66.426,-46.872,-179.004,5.686,148.706
C02460=1207.797,66.176,-46.855,-179.006,5.685,148.706
C02461=1207.802,65.927,-46.838,-179.009,5.684,148.707
C02462=1207.807,65.677,-46.821,-179.012,5.684,148.708
C02463=1207.812,65.427,-46.804,-179.014,5.682,148.708
C02464=1207.817,65.179,-46.788,-179.017,5.682,148.709
C02465=1207.822,64.929,-46.771,-179.020,5.681,148.710
C02466=1207.826,64.680,-46.753,-179.022,5.680,148.710
C02467=1207.831,64.430,-46.737,-179.024,5.679,148.711
C02468=1207.837,64.181,-46.720,-179.027,5.679,148.711
C02469=1207.841,63.932,-46.703,-179.030,5.678,148.712
C02470=1207.846,63.682,-46.686,-179.032,5.677,148.712
C02471=1207.851,63.433,-46.669,-179.035,5.676,148.713
C02472=1207.856,63.184,-46.653,-179.038,5.676,148.714
C02473=1207.861,62.934,-46.636,-179.040,5.675,148.714
C02474=1207.866,62.684,-46.619,-179.042,5.674,148.715
C02475=1207.872,62.435,-46.602,-179.045,5.674,148.715
C02476=1207.876,62.186,-46.585,-179.048,5.673,148.716
C02477=1207.880,61.936,-46.569,-179.050,5.672,148.717
C02478=1207.886,61.687,-46.551,-179.053,5.671,148.717
C02479=1207.891,61.438,-46.535,-179.056,5.670,148.718
C02480=1207.895,61.188,-46.518,-179.058,5.670,148.719
C02481=1207.900,60.939,-46.501,-179.060,5.669,148.719
C02482=1207.906,60.690,-46.485,-179.063,5.668,148.720
C02483=1207.910,60.440,-46.468,-179.066,5.668,148.720
C02484=1207.915,60.191,-46.451,-179.068,5.667,148.721
C02485=1207.920,59.942,-46.435,-179.070,5.666,148.721
C02486=1207.925,59.692,-46.418,-179.073,5.666,148.722
C02487=1207.930,59.442,-46.401,-179.076,5.664,148.723
C02488=1207.935,59.194,-46.384,-179.078,5.663,148.723
C02489=1207.940,58.944,-46.368,-179.081,5.663,148.724
C02490=1207.945,58.694,-46.350,-179.084,5.662,148.725
C02491=1207.950,58.445,-46.335,-179.086,5.662,148.725
C02492=1207.955,58.196,-46.318,-179.088,5.661,148.726
C02493=1207.960,57.946,-46.301,-179.091,5.660,148.726
C02494=1207.965,57.697,-46.285,-179.094,5.660,148.727
C02495=1207.969,57.447,-46.268,-179.096,5.659,148.728
C02496=1207.974,57.198,-46.251,-179.099,5.657,148.728
C02497=1207.980,56.949,-46.234,-179.102,5.657,148.729
C02498=1207.985,56.699,-46.218,-179.104,5.656,148.729
C02499=1207.990,56.450,-46.202,-179.107,5.656,148.730
C02500=1207.994,56.200,-46.185,-179.109,5.655,148.730
C02501=1207.999,55.951,-46.168,-179.112,5.654,148.731
C02502=1208.004,55.702,-46.152,-179.114,5.654,148.732
C02503=1208.009,55.433,-46.134,-179.117,5.653,148.732
C02504=1208.015,55.165,-46.117,-179.120,5.652,148.733
C02505=1208.021,54.896,-46.099,-179.123,5.651,148.734
C02506=1208.026,54.628,-46.081,-179.125,5.651,148.734
C02507=1208.031,54.379,-46.065,-179.128,5.650,148.735
C02508=1208.035,54.129,-46.048,-179.130,5.649,148.736
C02509=1208.040,53.879,-46.032,-179.133,5.649,148.736
C02510=1208.046,53.630,-46.015,-179.136,5.648,148.737
C02511=1208.050,53.381,-45.999,-179.138,5.646,148.737
C02512=1208.056,53.131,-45.983,-179.141,5.646,148.738
C02513=1208.060,52.882,-45.966,-179.144,5.645,148.739
C02514=1208.065,52.633,-45.950,-179.146,5.645,148.739
C02515=1208.070,52.383,-45.933,-179.148,5.644,148.740
C02516=1208.074,52.133,-45.917,-179.151,5.643,148.740
C02517=1208.080,51.885,-45.901,-179.154,5.643,148.741
C02518=1208.085,51.634,-45.884,-179.156,5.642,148.742
C02519=1208.090,51.385,-45.868,-179.158,5.641,148.742
C02520=1208.095,51.136,-45.852,-179.161,5.641,148.743
C02521=1208.100,50.886,-45.836,-179.164,5.640,148.744
C02522=1208.104,50.637,-45.819,-179.166,5.640,148.744
C02523=1208.110,50.388,-45.803,-179.168,5.639,148.745
C02524=1208.114,50.138,-45.787,-179.171,5.638,148.745
C02525=1208.119,49.889,-45.771,-179.174,5.638,148.746
C02526=1208.124,49.639,-45.755,-179.177,5.636,148.747
C02527=1208.129,49.390,-45.738,-179.180,5.636,148.747
C02528=1208.134,49.141,-45.722,-179.182,5.635,148.748
C02529=1208.139,48.892,-45.706,-179.184,5.634,148.748
C02530=1208.144,48.642,-45.689,-179.187,5.634,148.749
C02531=1208.150,48.392,-45.673,-179.190,5.633,148.750
C02532=1208.154,48.143,-45.657,-179.192,5.632,148.750
C02533=1208.160,47.893,-45.641,-179.194,5.632,148.751
C02534=1208.164,47.644,-45.624,-179.197,5.631,148.752
C02535=1208.169,47.395,-45.609,-179.200,5.631,148.752
C02536=1208.174,47.145,-45.592,-179.202,5.630,148.753
C02537=1208.179,46.896,-45.577,-179.204,5.629,148.753
C02538=1208.184,46.646,-45.560,-179.207,5.629,148.754
C02539=1208.189,46.397,-45.544,-179.210,5.628,148.755
C02540=1208.194,46.147,-45.528,-179.212,5.628,148.755
C02541=1208.199,45.898,-45.512,-179.215,5.627,148.756
C02542=1208.204,45.648,-45.495,-179.217,5.626,148.757
C02543=1208.209,45.399,-45.480,-179.220,5.626,148.757
C02544=1208.213,45.150,-45.463,-179.222,5.625,148.758
C02545=1208.219,44.900,-45.448,-179.225,5.624,148.758
C02546=1208.223,44.651,-45.433,-179.227,5.624,148.759
C02547=1208.228,44.402,-45.416,-179.230,5.622,148.760
C02548=1208.233,44.152,-45.400,-179.233,5.622,148.760
C02549=1208.238,43.903,-45.384,-179.236,5.621,148.761
C02550=1208.243,43.653,-45.368,-179.238,5.620,148.761
C02551=1208.248,43.403,-45.352,-179.241,5.620,148.762
C02552=1208.253,43.154,-45.336,-179.243,5.619,148.763
C02553=1208.258,42.905,-45.320,-179.246,5.619,148.763
C02554=1208.263,42.655,-45.304,-179.248,5.618,148.764
C02555=1208.268,42.406,-45.288,-179.251,5.617,148.765
C02556=1208.273,42.156,-45.272,-179.253,5.617,148.765
C02557=1208.278,41.907,-45.256,-179.256,5.616,148.766
C02558=1208.283,41.658,-45.241,-179.259,5.616,148.767
C02559=1208.288,41.408,-45.225,-179.261,5.615,148.767
C02560=1208.293,41.159,-45.209,-179.263,5.614,148.768
C02561=1208.298,40.910,-45.193,-179.266,5.614,148.768
C02562=1208.303,40.660,-45.177,-179.269,5.613,148.769
C02563=1208.308,40.410,-45.161,-179.271,5.613,148.770
C02564=1208.313,40.160,-45.145,-179.273,5.612,148.770
C02565=1208.317,39.912,-45.130,-179.276,5.611,148.771
C02566=1208.323,39.662,-45.114,-179.279,5.611,148.772
C02567=1208.328,39.412,-45.098,-179.281,5.610,148.772
C02568=1208.333,39.163,-45.083,-179.284,5.610,148.773
C02569=1208.338,38.913,-45.067,-179.286,5.609,148.773
C02570=1208.343,38.664,-45.050,-179.289,5.608,148.774
C02571=1208.347,38.415,-45.035,-179.291,5.608,148.775
C02572=1208.353,38.165,-45.020,-179.294,5.607,148.775
C02573=1208.358,37.915,-45.004,-179.297,5.607,148.776
C02574=1208.363,37.666,-44.988,-179.299,5.606,148.776
C02575=1208.368,37.417,-44.972,-179.301,5.605,148.777
C02576=1208.372,37.167,-44.956,-179.304,5.605,148.778
C02577=1208.378,36.918,-44.941,-179.307,5.604,148.778
C02578=1208.383,36.669,-44.925,-179.309,5.603,148.779
C02579=1208.388,36.418,-44.909,-179.312,5.603,148.780
C02580=1208.392,36.169,-44.894,-179.314,5.602,148.780
C02581=1208.398,35.920,-44.879,-179.317,5.602,148.781
C02582=1208.403,35.671,-44.862,-179.319,5.601,148.782
C02583=1208.408,35.421,-44.846,-179.322,5.600,148.782
C02584=1208.412,35.172,-44.832,-179.325,5.600,148.783
C02585=1208.418,34.923,-44.816,-179.327,5.599,148.783
C02586=1208.422,34.672,-44.800,-179.330,5.599,148.784
C02587=1208.428,34.423,-44.784,-179.332,5.598,148.785
C02588=1208.432,34.174,-44.769,-179.335,5.597,148.785
C02589=1208.438,33.925,-44.754,-179.337,5.597,148.786
C02590=1208.443,33.674,-44.738,-179.340,5.596,148.787
C02591=1208.447,33.425,-44.723,-179.342,5.595,148.787
C02592=1208.453,33.176,-44.707,-179.345,5.595,148.788
C02593=1208.458,32.927,-44.692,-179.348,5.594,148.789
C02594=1208.462,32.677,-44.676,-179.350,5.594,148.789
C02595=1208.468,32.427,-44.661,-179.352,5.593,148.790
C02596=1208.473,32.178,-44.645,-179.355,5.592,148.790
C02597=1208.478,31.929,-44.630,-179.358,5.592,148.791
C02598=1208.482,31.679,-44.614,-179.360,5.591,148.792
C02599=1208.488,31.429,-44.599,-179.363,5.591,148.792
C02600=1208.492,31.180,-44.584,-179.366,5.590,148.793
C02601=1208.498,30.931,-44.568,-179.368,5.589,148.794
C02602=1208.502,30.681,-44.553,-179.370,5.589,148.794
C02603=1208.507,30.432,-44.537,-179.372,5.589,148.795
C02604=1208.513,30.182,-44.521,-179.375,5.589,148.796
C02605=1208.517,29.933,-44.506,-179.378,5.588,148.796
C02606=1208.523,29.684,-44.491,-179.380,5.587,148.797
C02607=1208.528,29.414,-44.474,-179.383,5.587,148.798
C02608=1208.533,29.146,-44.458,-179.386,5.586,148.798
C02609=1208.539,28.877,-44.442,-179.389,5.585,148.799
C02610=1208.543,28.609,-44.425,-179.392,5.585,148.800
C02611=1208.549,28.359,-44.410,-179.394,5.584,148.800
C02612=1208.554,28.110,-44.394,-179.396,5.583,148.801
C02613=1208.559,27.860,-44.380,-179.399,5.583,148.801
C02614=1208.564,27.611,-44.364,-179.402,5.582,148.802
C02615=1208.569,27.361,-44.349,-179.404,5.582,148.803
C02616=1208.574,27.111,-44.333,-179.407,5.581,148.803
C02617=1208.579,26.862,-44.318,-179.408,5.581,148.804
C02618=1208.584,26.613,-44.303,-179.411,5.581,148.805
C02619=1208.589,26.363,-44.288,-179.414,5.580,148.805
C02620=1208.594,26.114,-44.273,-179.416,5.580,148.806
C02621=1208.598,25.864,-44.257,-179.419,5.579,148.807
C02622=1208.604,25.615,-44.242,-179.422,5.578,148.807
C02623=1208.609,25.365,-44.227,-179.424,5.578,148.808
C02624=1208.614,25.116,-44.212,-179.426,5.577,148.808
C02625=1208.619,24.866,-44.197,-179.429,5.577,148.809
C02626=1208.624,24.617,-44.181,-179.432,5.576,148.810
C02627=1208.629,24.367,-44.167,-179.434,5.576,148.811
C02628=1208.634,24.117,-44.151,-179.437,5.575,148.811
C02629=1208.639,23.868,-44.136,-179.440,5.574,148.812
C02630=1208.644,23.619,-44.120,-179.442,5.574,148.812
C02631=1208.649,23.369,-44.106,-179.445,5.573,148.813
C02632=1208.654,23.120,-44.091,-179.447,5.573,148.814
C02633=1208.659,22.871,-44.076,-179.449,5.573,148.814
C02634=1208.664,22.621,-44.061,-179.452,5.572,148.815
C02635=1208.669,22.371,-44.046,-179.455,5.572,148.816
C02636=1208.674,22.122,-44.031,-179.457,5.571,148.816
C02637=1208.680,21.872,-44.016,-179.459,5.570,148.817
C02638=1208.684,21.623,-44.001,-179.462,5.570,148.818
C02639=1208.689,21.373,-43.985,-179.465,5.569,148.818
C02640=1208.694,21.123,-43.971,-179.467,5.569,148.819
C02641=1208.699,20.874,-43.956,-179.470,5.568,148.820
C02642=1208.704,20.624,-43.941,-179.472,5.567,148.820
C02643=1208.709,20.375,-43.926,-179.475,5.567,148.821
C02644=1208.714,20.126,-43.911,-179.477,5.566,148.821
C02645=1208.719,19.876,-43.896,-179.480,5.566,148.822
C02646=1208.724,19.627,-43.881,-179.482,5.566,148.823
C02647=1208.730,19.377,-43.866,-179.485,5.566,148.823
C02648=1208.734,19.128,-43.851,-179.487,5.565,148.824
C02649=1208.739,18.878,-43.837,-179.490,5.564,148.825
C02650=1208.745,18.629,-43.821,-179.492,5.564,148.825
C02651=1208.749,18.380,-43.806,-179.495,5.563,148.826
C02652=1208.754,18.130,-43.792,-179.497,5.563,148.827
C02653=1208.760,17.881,-43.776,-179.500,5.562,148.827
C02654=1208.765,17.631,-43.762,-179.503,5.562,148.828
C02655=1208.769,17.382,-43.747,-179.505,5.561,148.829
C02656=1208.774,17.132,-43.733,-179.508,5.560,148.829
C02657=1208.780,16.883,-43.717,-179.510,5.561,148.830
C02658=1208.785,16.633,-43.703,-179.512,5.560,148.830
C02659=1208.789,16.384,-43.688,-179.515,5.559,148.831
C02660=1208.795,16.134,-43.673,-179.518,5.559,148.832
C02661=1208.800,15.884,-43.659,-179.520,5.558,148.833
C02662=1208.804,15.635,-43.644,-179.523,5.558,148.833
C02663=1208.809,15.385,-43.630,-179.525,5.557,148.834
C02664=1208.815,15.136,-43.614,-179.528,5.557,148.834
C02665=1208.820,14.886,-43.600,-179.530,5.556,148.835
C02666=1208.824,14.637,-43.585,-179.533,5.556,148.836
C02667=1208.829,14.387,-43.570,-179.535,5.556,148.836
C02668=1208.835,14.137,-43.556,-179.538,5.555,148.837
C02669=1208.840,13.888,-43.541,-179.540,5.555,148.838
C02670=1208.845,13.639,-43.526,-179.543,5.554,148.838
C02671=1208.849,13.389,-43.511,-179.545,5.553,148.839
C02672=1208.855,13.139,-43.496,-179.548,5.553,148.840
C02673=1208.860,12.890,-43.482,-179.550,5.552,148.840
C02674=1208.865,12.641,-43.467,-179.553,5.552,148.841
C02675=1208.870,12.391,-43.453,-179.556,5.551,148.842
C02676=1208.875,12.141,-43.439,-179.558,5.552,148.842
C02677=1208.880,11.892,-43.423,-179.560,5.551,148.843
C02678=1208.885,11.642,-43.409,-179.563,5.550,148.843
C02679=1208.890,11.392,-43.394,-179.565,5.550,148.844
C02680=1208.894,11.143,-43.379,-179.568,5.549,148.845
C02681=1208.900,10.894,-43.366,-179.571,5.549,148.846
C02682=1208.905,10.645,-43.351,-179.573,5.548,148.846
C02683=1208.911,10.395,-43.336,-179.576,5.548,148.847
C02684=1208.915,10.145,-43.321,-179.577,5.548,148.847
C02685=1208.920,9.896,-43.307,-179.580,5.547,148.848
C02686=1208.925,9.646,-43.293,-179.583,5.547,148.849
C02687=1208.930,9.396,-43.279,-179.585,5.546,148.849
C02688=1208.935,9.147,-43.264,-179.588,5.546,148.850
C02689=1208.940,8.898,-43.249,-179.591,5.545,148.851
C02690=1208.945,8.648,-43.234,-179.593,5.545,148.851
C02691=1208.951,8.399,-43.220,-179.595,5.545,148.852
C02692=1208.956,8.149,-43.206,-179.598,5.544,148.853
C02693=1208.961,7.900,-43.191,-179.600,5.543,148.853
C02694=1208.966,7.650,-43.177,-179.603,5.543,148.854
C02695=1208.971,7.400,-43.163,-179.606,5.542,148.855
C02696=1208.975,7.151,-43.148,-179.608,5.542,148.855
C02697=1208.980,6.901,-43.134,-179.611,5.541,148.856
C02698=1208.985,6.652,-43.119,-179.613,5.542,148.857
C02699=1208.991,6.403,-43.105,-179.616,5.541,148.857
C02700=1208.996,6.153,-43.091,-179.618,5.540,148.858
C02701=1209.001,5.903,-43.077,-179.620,5.540,148.859
C02702=1209.006,5.654,-43.062,-179.623,5.539,148.859
C02703=1209.010,5.404,-43.048,-179.626,5.539,148.860
C02704=1209.015,5.154,-43.034,-179.628,5.538,148.861
C02705=1209.022,4.905,-43.019,-179.630,5.539,148.861
C02706=1209.027,4.655,-43.005,-179.633,5.538,148.862
C02707=1209.031,4.406,-42.990,-179.636,5.538,148.863
C02708=1209.036,4.156,-42.976,-179.638,5.537,148.863
C02709=1209.041,3.907,-42.961,-179.641,5.536,148.864
C02710=1209.046,3.657,-42.947,-179.643,5.536,148.865
C02711=1209.052,3.388,-42.933,-179.646,5.535,148.865
C02712=1209.057,3.119,-42.917,-179.649,5.535,148.866
C02713=1209.063,2.850,-42.902,-179.651,5.534,148.867
C02714=1209.068,2.581,-42.886,-179.654,5.534,148.867
C02715=1209.073,2.332,-42.872,-179.656,5.534,148.868
C02716=1209.078,2.082,-42.858,-179.659,5.534,148.869
C02717=1209.083,1.833,-42.844,-179.661,5.533,148.869
C02718=1209.088,1.583,-42.829,-179.664,5.533,148.870
C02719=1209.093,1.333,-42.815,-179.667,5.532,148.871
C02720=1209.098,1.084,-42.801,-179.669,5.531,148.871
C02721=1209.104,0.835,-42.787,-179.671,5.532,148.872
C02722=1209.109,0.585,-42.773,-179.674,5.531,148.873
C02723=1209.113,0.336,-42.759,-179.677,5.531,148.873
C02724=1209.118,0.085,-42.745,-179.679,5.530,148.874
C02725=1209.124,-0.164,-42.732,-179.681,5.529,148.875
C02726=1209.129,-0.413,-42.717,-179.684,5.529,148.875
C02727=1209.134,-0.663,-42.703,-179.686,5.529,148.876
C02728=1209.139,-0.913,-42.689,-179.689,5.529,148.877
C02729=1209.144,-1.162,-42.675,-179.691,5.528,148.877
C02730=1209.149,-1.412,-42.661,-179.694,5.528,148.878
C02731=1209.154,-1.661,-42.646,-179.697,5.527,148.879
C02732=1209.159,-1.911,-42.632,-179.699,5.526,148.879
C02733=1209.164,-2.160,-42.619,-179.701,5.527,148.880
C02734=1209.169,-2.409,-42.604,-179.704,5.526,148.881
C02735=1209.174,-2.660,-42.591,-179.706,5.526,148.881
C02736=1209.180,-2.909,-42.577,-179.709,5.525,148.882
C02737=1209.185,-3.158,-42.563,-179.712,5.525,148.883
C02738=1209.190,-3.408,-42.548,-179.714,5.525,148.883
C02739=1209.195,-3.658,-42.534,-179.716,5.524,148.884
C02740=1209.199,-3.907,-42.521,-179.719,5.524,148.885
C02741=1209.205,-4.157,-42.507,-179.721,5.523,148.885
C02742=1209.210,-4.407,-42.493,-179.724,5.523,148.886
C02743=1209.215,-4.656,-42.479,-179.726,5.522,148.887
C02744=1209.220,-4.905,-42.465,-179.728,5.522,148.887
C02745=1209.224,-5.155,-42.451,-179.731,5.522,148.888
C02746=1209.230,-5.404,-42.438,-179.734,5.521,148.889
C02747=1209.235,-5.654,-42.424,-179.736,5.521,148.889
C02748=1209.240,-5.904,-42.409,-179.739,5.520,148.890
C02749=1209.246,-6.153,-42.395,-179.741,5.521,148.891
C02750=1209.250,-6.403,-42.382,-179.743,5.520,148.891
C02751=1209.255,-6.653,-42.368,-179.746,5.519,148.892
C02752=1209.261,-6.902,-42.354,-179.749,5.519,148.893
C02753=1209.266,-7.152,-42.341,-179.751,5.518,148.893
C02754=1209.270,-7.401,-42.327,-179.753,5.519,148.894
C02755=1209.276,-7.650,-42.313,-179.756,5.518,148.895
C02756=1209.281,-7.900,-42.299,-179.759,5.518,148.895
C02757=1209.286,-8.150,-42.285,-179.761,5.517,148.896
C02758=1209.291,-8.399,-42.272,-179.764,5.517,148.897
C02759=1209.296,-8.649,-42.258,-179.766,5.517,148.897
C02760=1209.301,-8.899,-42.244,-179.768,5.516,148.898
C02761=1209.306,-9.148,-42.231,-179.771,5.516,148.899
C02762=1209.311,-9.397,-42.216,-179.774,5.515,148.899
C02763=1209.317,-9.647,-42.203,-179.776,5.515,148.900
C02764=1209.322,-9.897,-42.189,-179.778,5.515,148.901
C02765=1209.326,-10.147,-42.176,-179.781,5.514,148.901
C02766=1209.332,-10.396,-42.162,-179.784,5.514,148.902
C02767=1209.337,-10.646,-42.148,-179.786,5.514,148.903
C02768=1209.342,-10.895,-42.135,-179.788,5.514,148.903
C02769=1209.347,-11.145,-42.121,-179.791,5.513,148.904
C02770=1209.352,-11.395,-42.107,-179.793,5.512,148.905
C02771=1209.357,-11.644,-42.094,-179.796,5.512,148.905
C02772=1209.362,-11.893,-42.080,-179.798,5.511,148.906
C02773=1209.368,-12.143,-42.067,-179.801,5.512,148.907
C02774=1209.372,-12.392,-42.053,-179.803,5.511,148.907
C02775=1209.377,-12.643,-42.039,-179.806,5.511,148.908
C02776=1209.382,-12.891,-42.026,-179.809,5.510,148.909
C02777=1209.387,-13.142,-42.012,-179.811,5.511,148.909
C02778=1209.393,-13.391,-41.999,-179.813,5.510,148.910
C02779=1209.397,-13.641,-41.986,-179.815,5.509,148.911
C02780=1209.403,-13.890,-41.972,-179.818,5.509,148.911
C02781=1209.408,-14.140,-41.958,-179.820,5.509,148.912
C02782=1209.412,-14.389,-41.944,-179.823,5.509,148.913
C02783=1209.418,-14.639,-41.931,-179.825,5.508,148.913
C02784=1209.422,-14.889,-41.918,-179.828,5.508,148.914
C02785=1209.428,-15.138,-41.904,-179.831,5.507,148.915
C02786=1209.432,-15.388,-41.891,-179.833,5.507,148.915
C02787=1209.438,-15.637,-41.878,-179.836,5.507,148.916
C02788=1209.443,-15.887,-41.863,-179.838,5.506,148.917
C02789=1209.448,-16.136,-41.851,-179.840,5.506,148.917
C02790=1209.453,-16.386,-41.836,-179.842,5.506,148.918
C02791=1209.458,-16.635,-41.824,-179.845,5.505,148.919
C02792=1209.464,-16.886,-41.810,-179.848,5.505,148.919
C02793=1209.468,-17.134,-41.797,-179.850,5.504,148.920
C02794=1209.474,-17.385,-41.783,-179.852,5.505,148.921
C02795=1209.479,-17.633,-41.770,-179.855,5.504,148.921
C02796=1209.484,-17.884,-41.756,-179.858,5.504,148.922
C02797=1209.489,-18.133,-41.744,-179.860,5.503,148.923
C02798=1209.494,-18.383,-41.730,-179.863,5.504,148.923
C02799=1209.499,-18.632,-41.717,-179.865,5.503,148.924
C02800=1209.504,-18.882,-41.703,-179.867,5.502,148.925
C02801=1209.509,-19.131,-41.690,-179.870,5.502,148.925
C02802=1209.514,-19.381,-41.677,-179.872,5.502,148.926
C02803=1209.519,-19.631,-41.664,-179.875,5.502,148.927
C02804=1209.524,-19.880,-41.650,-179.877,5.501,148.927
C02805=1209.530,-20.130,-41.637,-179.880,5.501,148.928
C02806=1209.535,-20.379,-41.624,-179.882,5.501,148.929
C02807=1209.540,-20.629,-41.610,-179.885,5.501,148.930
C02808=1209.545,-20.878,-41.597,-179.887,5.500,148.930
C02809=1209.550,-21.128,-41.584,-179.890,5.499,148.931
C02810=1209.556,-21.377,-41.570,-179.892,5.500,148.931
C02811=1209.560,-21.627,-41.557,-179.894,5.499,148.932
C02812=1209.566,-21.877,-41.544,-179.897,5.499,148.933
C02813=1209.570,-22.127,-41.531,-179.900,5.498,148.933
C02814=1209.575,-22.376,-41.518,-179.902,5.498,148.934
C02815=1209.581,-22.646,-41.503,-179.904,5.498,148.935
C02816=1209.587,-22.915,-41.489,-179.907,5.497,148.936
C02817=1209.592,-23.184,-41.475,-179.910,5.497,148.936
C02818=1209.598,-23.454,-41.461,-179.913,5.497,148.937
C02819=1209.603,-23.704,-41.448,-179.915,5.496,148.938
C02820=1209.608,-23.954,-41.435,-179.917,5.496,148.938
C02821=1209.613,-24.203,-41.421,-179.920,5.496,148.939
C02822=1209.618,-24.452,-41.409,-179.922,5.495,148.940
C02823=1209.623,-24.702,-41.395,-179.925,5.495,148.940
C02824=1209.628,-24.952,-41.383,-179.927,5.495,148.941
C02825=1209.633,-25.202,-41.370,-179.930,5.495,148.942
C02826=1209.639,-25.451,-41.356,-179.933,5.494,148.943
C02827=1209.644,-25.700,-41.343,-179.935,5.495,148.943
C02828=1209.649,-25.950,-41.330,-179.937,5.494,148.944
C02829=1209.654,-26.200,-41.317,-179.939,5.493,148.944
C02830=1209.659,-26.450,-41.304,-179.942,5.493,148.945
C02831=1209.664,-26.699,-41.291,-179.944,5.493,148.946
C02832=1209.670,-26.948,-41.278,-179.947,5.493,148.946
C02833=1209.674,-27.199,-41.265,-179.950,5.492,148.947
C02834=1209.679,-27.448,-41.253,-179.952,5.492,148.948
C02835=1209.685,-27.697,-41.239,-179.954,5.492,148.949
C02836=1209.689,-27.947,-41.226,-179.957,5.491,148.949
C02837=1209.694,-28.196,-41.213,-179.960,5.491,148.950
C02838=1209.700,-28.446,-41.200,-179.962,5.491,148.951
C02839=1209.705,-28.696,-41.187,-179.964,5.491,148.951
C02840=1209.710,-28.945,-41.174,-179.966,5.490,148.952
C02841=1209.715,-29.194,-41.162,-179.969,5.489,148.953
C02842=1209.720,-29.445,-41.148,-179.971,5.490,148.953
C02843=1209.725,-29.694,-41.136,-179.974,5.489,148.954
C02844=1209.731,-29.943,-41.123,-179.977,5.489,148.955
C02845=1209.736,-30.194,-41.109,-179.979,5.489,148.955
C02846=1209.741,-30.443,-41.097,-179.981,5.489,148.956
C02847=1209.746,-30.692,-41.084,-179.984,5.488,148.957
C02848=1209.751,-30.942,-41.071,-179.986,5.489,148.957
C02849=1209.756,-31.192,-41.059,-179.989,5.488,148.958
C02850=1209.762,-31.441,-41.045,-179.991,5.487,148.959
C02851=1209.766,-31.691,-41.032,-179.994,5.487,148.959
C02852=1209.771,-31.941,-41.020,-179.996,5.487,148.960
C02853=1209.776,-32.190,-41.007,-179.998,5.487,148.961
C02854=1209.782,-32.440,-40.994,179.999,5.486,148.961
C02855=1209.787,-32.690,-40.981,179.997,5.486,148.962
C02856=1209.792,-32.939,-40.969,179.994,5.486,148.963
C02857=1209.797,-33.189,-40.957,179.992,5.486,148.963
C02858=1209.802,-33.439,-40.944,179.989,5.485,148.964
C02859=1209.808,-33.689,-40.930,179.987,5.485,148.965
C02860=1209.813,-33.938,-40.918,179.984,5.485,148.966
C02861=1209.818,-34.187,-40.905,179.982,5.484,148.966
C02862=1209.822,-34.437,-40.892,179.980,5.484,148.967
C02863=1209.828,-34.687,-40.880,179.977,5.484,148.967
C02864=1209.833,-34.936,-40.867,179.975,5.483,148.968
C02865=1209.839,-35.185,-40.854,179.973,5.484,148.969
C02866=1209.843,-35.436,-40.842,179.970,5.483,148.970
C02867=1209.849,-35.685,-40.829,179.967,5.483,148.970
C02868=1209.854,-35.935,-40.816,179.965,5.483,148.971
C02869=1209.859,-36.184,-40.804,179.963,5.483,148.972
C02870=1209.863,-36.434,-40.791,179.960,5.482,148.972
C02871=1209.868,-36.683,-40.778,179.958,5.481,148.973
C02872=1209.874,-36.933,-40.766,179.956,5.482,148.973
C02873=1209.880,-37.183,-40.753,179.953,5.481,148.974
C02874=1209.885,-37.432,-40.741,179.950,5.481,148.975
C02875=1209.889,-37.682,-40.728,179.948,5.481,148.976
C02876=1209.895,-37.932,-40.716,179.946,5.481,148.976
C02877=1209.900,-38.182,-40.703,179.943,5.480,148.977
C02878=1209.905,-38.431,-40.691,179.941,5.480,148.978
C02879=1209.910,-38.680,-40.678,179.938,5.480,148.978
C02880=1209.915,-38.931,-40.666,179.935,5.480,148.979
C02881=1209.920,-39.180,-40.653,179.933,5.480,148.980
C02882=1209.925,-39.429,-40.640,179.931,5.479,148.980
C02883=1209.930,-39.679,-40.628,179.929,5.479,148.981
C02884=1209.936,-39.929,-40.616,179.926,5.479,148.982
C02885=1209.940,-40.179,-40.603,179.924,5.478,148.982
C02886=1209.945,-40.428,-40.590,179.921,5.478,148.983
C02887=1209.951,-40.677,-40.578,179.919,5.478,148.984
C02888=1209.957,-40.928,-40.565,179.916,5.478,148.984
C02889=1209.962,-41.177,-40.553,179.914,5.477,148.985
C02890=1209.967,-41.426,-40.540,179.912,5.478,148.986
C02891=1209.972,-41.677,-40.528,179.909,5.477,148.987
C02892=1209.977,-41.926,-40.515,179.907,5.476,148.987
C02893=1209.982,-42.176,-40.503,179.905,5.477,148.988
C02894=1209.987,-42.425,-40.491,179.902,5.476,148.988
C02895=1209.993,-42.675,-40.478,179.899,5.476,148.989
C02896=1209.998,-42.925,-40.466,179.897,5.476,148.990
C02897=1210.002,-43.174,-40.454,179.895,5.476,148.991
C02898=1210.007,-43.424,-40.441,179.892,5.475,148.991
C02899=1210.012,-43.674,-40.429,179.890,5.476,148.992
C02900=1210.017,-43.923,-40.417,179.887,5.475,148.993
C02901=1210.023,-44.173,-40.405,179.885,5.475,148.993
C02902=1210.028,-44.422,-40.392,179.883,5.475,148.994
C02903=1210.033,-44.672,-40.380,179.880,5.474,148.995
C02904=1210.039,-44.922,-40.368,179.878,5.474,148.995
C02905=1210.044,-45.171,-40.355,179.876,5.474,148.996
C02906=1210.049,-45.421,-40.343,179.873,5.474,148.997
C02907=1210.054,-45.671,-40.330,179.870,5.473,148.997
C02908=1210.059,-45.921,-40.319,179.868,5.473,148.998
C02909=1210.064,-46.170,-40.306,179.866,5.473,148.999
C02910=1210.070,-46.420,-40.294,179.863,5.472,148.999
C02911=1210.075,-46.669,-40.281,179.861,5.473,149.000
C02912=1210.080,-46.919,-40.270,179.859,5.472,149.001
C02913=1210.085,-47.168,-40.258,179.856,5.472,149.001
C02914=1210.090,-47.418,-40.246,179.854,5.472,149.002
C02915=1210.095,-47.667,-40.233,179.851,5.471,149.003
C02916=1210.101,-47.917,-40.221,179.849,5.471,149.003
C02917=1210.106,-48.167,-40.209,179.846,5.471,149.004
C02918=1210.111,-48.417,-40.197,179.844,5.471,149.005
C02919=1210.116,-48.686,-40.183,179.841,5.470,149.006
C02920=1210.121,-48.957,-40.170,179.839,5.471,149.006
C02921=1210.127,-49.226,-40.157,179.836,5.470,149.007
C02922=1210.133,-49.497,-40.144,179.834,5.470,149.008
C02923=1210.138,-49.746,-40.132,179.831,5.469,149.008
C02924=1210.143,-49.996,-40.120,179.829,5.470,149.009
C02925=1210.148,-50.245,-40.107,179.826,5.469,149.010
C02926=1210.154,-50.495,-40.096,179.824,5.470,149.010
C02927=1210.159,-50.745,-40.084,179.822,5.469,149.011
C02928=1210.164,-50.994,-40.072,179.819,5.469,149.012
C02929=1210.169,-51.244,-40.060,179.817,5.469,149.013
C02930=1210.174,-51.493,-40.047,179.814,5.468,149.013
C02931=1210.180,-51.743,-40.035,179.812,5.468,149.014
C02932=1210.185,-51.993,-40.023,179.810,5.468,149.014
C02933=1210.189,-52.242,-40.011,179.807,5.468,149.015
C02934=1210.195,-52.492,-40.000,179.805,5.467,149.016
C02935=1210.200,-52.742,-39.988,179.802,5.467,149.017
C02936=1210.205,-52.992,-39.975,179.800,5.467,149.017
C02937=1210.211,-53.241,-39.963,179.798,5.467,149.018
C02938=1210.215,-53.491,-39.952,179.795,5.467,149.019
C02939=1210.221,-53.740,-39.939,179.792,5.466,149.019
C02940=1210.226,-53.990,-39.927,179.790,5.467,149.020
C02941=1210.231,-54.240,-39.915,179.788,5.466,149.021
C02942=1210.236,-54.489,-39.903,179.785,5.465,149.021
C02943=1210.241,-54.739,-39.892,179.783,5.466,149.022
C02944=1210.247,-54.989,-39.880,179.781,5.465,149.023
C02945=1210.251,-55.239,-39.868,179.779,5.466,149.023
C02946=1210.257,-55.488,-39.856,179.776,5.465,149.024
C02947=1210.262,-55.738,-39.844,179.773,5.465,149.025
C02948=1210.267,-55.988,-39.832,179.771,5.465,149.025
C02949=1210.272,-56.238,-39.821,179.768,5.465,149.026
C02950=1210.277,-56.487,-39.808,179.766,5.464,149.027
C02951=1210.283,-56.737,-39.796,179.764,5.464,149.027
C02952=1210.287,-56.986,-39.785,179.762,5.464,149.028
C02953=1210.293,-57.236,-39.773,179.759,5.464,149.029
C02954=1210.298,-57.486,-39.760,179.757,5.464,149.029
C02955=1210.303,-57.735,-39.749,179.754,5.463,149.030
C02956=1210.308,-57.985,-39.737,179.752,5.464,149.031
C02957=1210.313,-58.235,-39.725,179.749,5.463,149.032
C02958=1210.318,-58.485,-39.714,179.747,5.463,149.032
C02959=1210.324,-58.735,-39.702,179.745,5.463,149.033
C02960=1210.329,-58.983,-39.690,179.742,5.462,149.033
C02961=1210.334,-59.233,-39.679,179.740,5.462,149.034
C02962=1210.339,-59.483,-39.667,179.738,5.462,149.035
C02963=1210.344,-59.733,-39.656,179.735,5.462,149.036
C02964=1210.350,-59.983,-39.644,179.733,5.462,149.036
C02965=1210.355,-60.232,-39.632,179.730,5.461,149.037
C02966=1210.360,-60.482,-39.620,179.728,5.462,149.038
C02967=1210.365,-60.731,-39.608,179.726,5.461,149.038
C02968=1210.370,-60.981,-39.596,179.723,5.461,149.039
C02969=1210.375,-61.231,-39.585,179.721,5.461,149.040
C02970=1210.381,-61.480,-39.573,179.719,5.460,149.040
C02971=1210.386,-61.730,-39.562,179.717,5.461,149.041
C02972=1210.391,-61.980,-39.550,179.714,5.460,149.042
C02973=1210.396,-62.229,-39.539,179.711,5.460,149.042
C02974=1210.401,-62.479,-39.527,179.709,5.460,149.043
C02975=1210.407,-62.729,-39.515,179.706,5.460,149.044
C02976=1210.411,-62.979,-39.504,179.705,5.460,149.044
C02977=1210.417,-63.229,-39.492,179.702,5.459,149.045
C02978=1210.422,-63.478,-39.481,179.700,5.459,149.046
C02979=1210.427,-63.728,-39.469,179.697,5.459,149.046
C02980=1210.432,-63.977,-39.458,179.695,5.459,149.047
C02981=1210.438,-64.227,-39.446,179.693,5.459,149.048
C02982=1210.442,-64.477,-39.435,179.690,5.459,149.049
C02983=1210.448,-64.727,-39.423,179.687,5.458,149.049
C02984=1210.453,-64.976,-39.412,179.685,5.459,149.050
C02985=1210.458,-65.226,-39.400,179.683,5.458,149.050
C02986=1210.464,-65.476,-39.388,179.681,5.458,149.051
C02987=1210.469,-65.725,-39.377,179.678,5.458,149.052
C02988=1210.474,-65.975,-39.365,179.676,5.457,149.053
C02989=1210.479,-66.225,-39.353,179.674,5.458,149.053
C02990=1210.485,-66.474,-39.342,179.671,5.457,149.054
C02991=1210.489,-66.724,-39.331,179.669,5.457,149.055
C02992=1210.494,-66.973,-39.319,179.666,5.457,149.055
C02993=1210.499,-67.223,-39.307,179.664,5.456,149.056
C02994=1210.504,-67.473,-39.296,179.662,5.457,149.057
C02995=1210.510,-67.722,-39.285,179.659,5.456,149.057
C02996=1210.515,-67.972,-39.273,179.657,5.456,149.058
C02997=1210.520,-68.222,-39.261,179.654,5.456,149.059
C02998=1210.525,-68.472,-39.251,179.652,5.456,149.059
C02999=1210.531,-68.722,-39.239,179.650,5.456,149.060
C03000=1210.536,-68.971,-39.228,179.647,5.455,149.061
C03001=1210.541,-69.221,-39.216,179.645,5.455,149.061
C03002=1210.546,-69.470,-39.205,179.643,5.455,149.062
C03003=1210.552,-69.720,-39.193,179.641,5.455,149.063
C03004=1210.557,-69.969,-39.182,179.638,5.455,149.063
C03005=1210.562,-70.219,-39.172,179.635,5.454,149.064
C03006=1210.567,-70.469,-39.160,179.633,5.455,149.065
C03007=1210.572,-70.719,-39.148,179.631,5.454,149.065
C03008=1210.578,-70.968,-39.137,179.629,5.454,149.066
C03009=1210.583,-71.218,-39.126,179.626,5.454,149.067
C03010=1210.588,-71.468,-39.115,179.624,5.454,149.067
C03011=1210.593,-71.718,-39.103,179.622,5.454,149.068
C03012=1210.598,-71.967,-39.092,179.619,5.453,149.069
C03013=1210.604,-72.217,-39.080,179.617,5.454,149.070
C03014=1210.609,-72.467,-39.069,179.614,5.453,149.070
C03015=1210.614,-72.717,-39.058,179.612,5.454,149.071
C03016=1210.620,-72.966,-39.047,179.610,5.453,149.071
C03017=1210.624,-73.216,-39.036,179.607,5.452,149.072
C03018=1210.629,-73.465,-39.024,179.605,5.453,149.073
C03019=1210.635,-73.715,-39.014,179.602,5.452,149.074
C03020=1210.640,-73.965,-39.002,179.600,5.453,149.074
C03021=1210.645,-74.214,-38.991,179.598,5.452,149.075
C03022=1210.651,-74.464,-38.979,179.596,5.453,149.076
C03023=1210.656,-74.735,-38.967,179.593,5.452,149.076
C03024=1210.661,-75.005,-38.956,179.590,5.452,149.077
C03025=1210.667,-75.276,-38.944,179.588,5.452,149.078
C03026=1210.673,-75.547,-38.931,179.585,5.452,149.078
C03027=1210.678,-75.796,-38.920,179.583,5.451,149.079
C03028=1210.684,-76.046,-38.909,179.581,5.452,149.080
C03029=1210.689,-76.296,-38.898,179.578,5.451,149.081
C03030=1210.693,-76.545,-38.887,179.576,5.451,149.081
C03031=1210.700,-76.795,-38.876,179.574,5.451,149.082
C03032=1210.704,-77.045,-38.865,179.571,5.450,149.083
C03033=1210.709,-77.294,-38.853,179.569,5.451,149.083
C03034=1210.715,-77.544,-38.843,179.566,5.450,149.084
C03035=1210.720,-77.794,-38.831,179.564,5.450,149.085
C03036=1210.725,-78.043,-38.820,179.562,5.450,149.085
C03037=1210.731,-78.293,-38.810,179.560,5.450,149.086
C03038=1210.735,-78.543,-38.798,179.557,5.450,149.087
C03039=1210.741,-78.793,-38.787,179.555,5.450,149.087
C03040=1210.746,-79.042,-38.776,179.553,5.450,149.088
C03041=1210.751,-79.292,-38.765,179.550,5.449,149.089
C03042=1210.756,-79.542,-38.754,179.548,5.449,149.089
C03043=1210.762,-79.791,-38.743,179.545,5.449,149.090
C03044=1210.767,-80.041,-38.732,179.544,5.449,149.091
C03045=1210.772,-80.290,-38.721,179.541,5.449,149.091
C03046=1210.777,-80.541,-38.711,179.539,5.449,149.092
C03047=1210.782,-80.790,-38.700,179.536,5.448,149.093
C03048=1210.788,-81.040,-38.689,179.534,5.449,149.093
C03049=1210.793,-81.290,-38.678,179.531,5.448,149.094
C03050=1210.798,-81.540,-38.667,179.529,5.448,149.095
C03051=1210.803,-81.789,-38.656,179.527,5.448,149.095
C03052=1210.808,-82.039,-38.645,179.524,5.448,149.096
C03053=1210.814,-82.288,-38.634,179.522,5.448,149.097
C03054=1210.819,-82.539,-38.623,179.520,5.447,149.097
C03055=1210.824,-82.788,-38.612,179.518,5.448,149.098
C03056=1210.830,-83.038,-38.602,179.515,5.447,149.099
C03057=1210.834,-83.287,-38.591,179.513,5.447,149.099
C03058=1210.840,-83.537,-38.580,179.511,5.447,149.100
C03059=1210.845,-83.787,-38.569,179.509,5.447,149.101
C03060=1210.851,-84.036,-38.558,179.506,5.447,149.101
C03061=1210.856,-84.286,-38.547,179.503,5.446,149.102
C03062=1210.861,-84.536,-38.536,179.501,5.447,149.103
C03063=1210.866,-84.785,-38.525,179.499,5.446,149.103
C03064=1210.871,-85.035,-38.515,179.497,5.446,149.104
C03065=1210.876,-85.285,-38.505,179.494,5.446,149.105
C03066=1210.881,-85.535,-38.493,179.492,5.446,149.105
C03067=1210.887,-85.784,-38.483,179.489,5.446,149.106
C03068=1210.891,-86.034,-38.472,179.487,5.446,149.107
C03069=1210.897,-86.284,-38.461,179.485,5.445,149.107
C03070=1210.903,-86.534,-38.451,179.483,5.446,149.108
C03071=1210.907,-86.784,-38.439,179.480,5.445,149.109
C03072=1210.913,-87.033,-38.429,179.478,5.446,149.110
C03073=1210.918,-87.283,-38.418,179.476,5.445,149.110
C03074=1210.923,-87.532,-38.408,179.473,5.445,149.111
C03075=1210.928,-87.782,-38.397,179.471,5.445,149.111
C03076=1210.934,-88.031,-38.386,179.469,5.444,149.112
C03077=1210.939,-88.282,-38.375,179.467,5.445,149.113
C03078=1210.944,-88.531,-38.365,179.464,5.444,149.114
C03079=1210.949,-88.781,-38.354,179.462,5.445,149.114
C03080=1210.955,-89.030,-38.344,179.459,5.444,149.115
C03081=1210.960,-89.281,-38.333,179.458,5.444,149.115
C03082=1210.965,-89.530,-38.322,179.455,5.444,149.116
C03083=1210.970,-89.780,-38.312,179.453,5.444,149.117
C03084=1210.975,-90.029,-38.301,179.450,5.444,149.118
C03085=1210.980,-90.280,-38.291,179.448,5.444,149.118
C03086=1210.986,-90.528,-38.280,179.445,5.444,149.119
C03087=1210.991,-90.779,-38.269,179.444,5.444,149.119
C03088=1210.996,-91.028,-38.259,179.441,5.443,149.120
C03089=1211.001,-91.279,-38.249,179.439,5.444,149.121
C03090=1211.007,-91.527,-38.238,179.436,5.443,149.122
C03091=1211.012,-91.778,-38.227,179.434,5.443,149.122
C03092=1211.017,-92.027,-38.217,179.432,5.443,149.123
C03093=1211.022,-92.277,-38.206,179.429,5.442,149.124
C03094=1211.027,-92.526,-38.195,179.427,5.443,149.124
C03095=1211.032,-92.777,-38.185,179.425,5.442,149.125
C03096=1211.038,-93.026,-38.175,179.423,5.443,149.126
C03097=1211.044,-93.276,-38.164,179.420,5.442,149.126
C03098=1211.049,-93.526,-38.154,179.418,5.442,149.127
C03099=1211.054,-93.775,-38.143,179.416,5.442,149.128
C03100=1211.059,-94.025,-38.132,179.413,5.442,149.128
C03101=1211.065,-94.275,-38.122,179.411,5.442,149.129
C03102=1211.070,-94.525,-38.112,179.409,5.442,149.130
C03103=1211.075,-94.774,-38.101,179.407,5.441,149.130
C03104=1211.080,-95.025,-38.091,179.404,5.442,149.131
C03105=1211.085,-95.274,-38.080,179.402,5.441,149.132
C03106=1211.091,-95.523,-38.070,179.400,5.442,149.132
C03107=1211.095,-95.773,-38.060,179.397,5.441,149.133
C03108=1211.101,-96.023,-38.049,179.395,5.441,149.134
C03109=1211.106,-96.273,-38.039,179.393,5.441,149.134
C03110=1211.111,-96.522,-38.029,179.391,5.441,149.135
C03111=1211.117,-96.772,-38.018,179.388,5.441,149.136
C03112=1211.122,-97.022,-38.008,179.386,5.441,149.136
C03113=1211.128,-97.272,-37.998,179.383,5.441,149.137
C03114=1211.132,-97.521,-37.986,179.382,5.441,149.138
C03115=1211.138,-97.771,-37.976,179.379,5.440,149.138
C03116=1211.143,-98.020,-37.967,179.377,5.441,149.139
C03117=1211.148,-98.270,-37.956,179.374,5.440,149.140
C03118=1211.153,-98.520,-37.946,179.372,5.441,149.140
C03119=1211.158,-98.770,-37.935,179.370,5.440,149.141
C03120=1211.164,-99.020,-37.925,179.368,5.440,149.142
C03121=1211.170,-99.269,-37.915,179.365,5.440,149.142
C03122=1211.175,-99.520,-37.904,179.363,5.440,149.143
C03123=1211.179,-99.769,-37.895,179.360,5.440,149.144
C03124=1211.185,-100.018,-37.884,179.358,5.439,149.144
C03125=1211.190,-100.269,-37.874,179.356,5.439,149.145
C03126=1211.196,-100.518,-37.864,179.353,5.439,149.146
C03127=1211.201,-100.789,-37.853,179.351,5.439,149.146
C03128=1211.207,-101.061,-37.841,179.349,5.439,149.147
C03129=1211.213,-101.332,-37.831,179.347,5.439,149.148
C03130=1211.218,-101.603,-37.819,179.344,5.439,149.149
C03131=1211.223,-101.852,-37.809,179.341,5.438,149.149
C03132=1211.228,-102.103,-37.799,179.339,5.439,149.150
C03133=1211.234,-102.352,-37.789,179.337,5.438,149.150
C03134=1211.240,-102.602,-37.778,179.335,5.438,149.151
C03135=1211.244,-102.852,-37.768,179.332,5.438,149.152
C03136=1211.249,-103.101,-37.758,179.330,5.438,149.153
C03137=1211.255,-103.351,-37.748,179.327,5.438,149.153
C03138=1211.260,-103.602,-37.738,179.326,5.438,149.154
C03139=1211.265,-103.851,-37.729,179.323,5.437,149.154
C03140=1211.271,-104.100,-37.718,179.321,5.438,149.155
C03141=1211.276,-104.351,-37.708,179.318,5.437,149.156
C03142=1211.281,-104.600,-37.698,179.317,5.437,149.156
C03143=1211.286,-104.849,-37.688,179.314,5.437,149.157
C03144=1211.291,-105.100,-37.677,179.312,5.437,149.158
C03145=1211.297,-105.349,-37.667,179.309,5.437,149.159
C03146=1211.302,-105.599,-37.657,179.307,5.437,149.159
C03147=1211.308,-105.849,-37.648,179.306,5.437,149.160
C03148=1211.313,-106.099,-37.637,179.303,5.437,149.160
C03149=1211.318,-106.348,-37.627,179.301,5.437,149.161
C03150=1211.323,-106.598,-37.618,179.298,5.437,149.162
C03151=1211.328,-106.848,-37.607,179.297,5.437,149.162
C03152=1211.334,-107.097,-37.597,179.294,5.436,149.163
C03153=1211.339,-107.347,-37.588,179.292,5.437,149.164
C03154=1211.344,-107.597,-37.578,179.289,5.436,149.165
C03155=1211.349,-107.847,-37.567,179.287,5.437,149.165
C03156=1211.354,-108.096,-37.558,179.285,5.436,149.166
C03157=1211.360,-108.346,-37.547,179.283,5.436,149.166
C03158=1211.366,-108.596,-37.538,179.280,5.436,149.167
C03159=1211.370,-108.846,-37.528,179.278,5.436,149.168
C03160=1211.376,-109.096,-37.518,179.276,5.436,149.168
C03161=1211.381,-109.345,-37.507,179.274,5.436,149.169
C03162=1211.386,-109.594,-37.498,179.271,5.436,149.170
C03163=1211.391,-109.845,-37.488,179.269,5.436,149.170
C03164=1211.397,-110.095,-37.478,179.267,5.435,149.171
C03165=1211.402,-110.344,-37.468,179.265,5.435,149.172
C03166=1211.408,-110.594,-37.459,179.262,5.435,149.172
C03167=1211.413,-110.843,-37.449,179.260,5.435,149.173
C03168=1211.418,-111.094,-37.438,179.258,5.435,149.174
C03169=1211.423,-111.343,-37.428,179.256,5.435,149.174
C03170=1211.428,-111.593,-37.419,179.253,5.435,149.175
C03171=1211.434,-111.843,-37.409,179.251,5.435,149.176
C03172=1211.438,-112.092,-37.399,179.249,5.434,149.176
C03173=1211.444,-112.343,-37.390,179.247,5.435,149.177
C03174=1211.450,-112.592,-37.379,179.244,5.434,149.178
C03175=1211.455,-112.841,-37.370,179.242,5.435,149.178
C03176=1211.460,-113.092,-37.360,179.240,5.434,149.179
C03177=1211.465,-113.341,-37.351,179.238,5.434,149.180
C03178=1211.470,-113.591,-37.340,179.235,5.434,149.180
C03179=1211.476,-113.841,-37.331,179.233,5.434,149.181
C03180=1211.481,-114.090,-37.321,179.231,5.434,149.181
C03181=1211.487,-114.340,-37.311,179.228,5.434,149.182
C03182=1211.492,-114.590,-37.302,179.226,5.434,149.183
C03183=1211.497,-114.840,-37.291,179.224,5.434,149.184
C03184=1211.502,-115.089,-37.282,179.222,5.434,149.184
C03185=1211.508,-115.339,-37.272,179.219,5.433,149.185
C03186=1211.513,-115.589,-37.263,179.217,5.434,149.186
C03187=1211.518,-115.839,-37.253,179.215,5.433,149.186
C03188=1211.523,-116.088,-37.244,179.213,5.433,149.187
C03189=1211.529,-116.338,-37.234,179.210,5.433,149.187
C03190=1211.533,-116.588,-37.224,179.208,5.433,149.188
C03191=1211.539,-116.838,-37.214,179.206,5.433,149.189
C03192=1211.544,-117.088,-37.205,179.204,5.433,149.189
C03193=1211.550,-117.337,-37.195,179.201,5.432,149.190
C03194=1211.555,-117.587,-37.186,179.199,5.433,149.191
C03195=1211.561,-117.836,-37.176,179.197,5.432,149.192
C03196=1211.566,-118.086,-37.167,179.195,5.432,149.192
C03197=1211.571,-118.337,-37.156,179.192,5.432,149.193
C03198=1211.576,-118.586,-37.147,179.190,5.432,149.193
C03199=1211.581,-118.836,-37.137,179.189,5.432,149.194
C03200=1211.587,-119.086,-37.128,179.186,5.432,149.195
C03201=1211.592,-119.335,-37.118,179.184,5.432,149.195
C03202=1211.597,-119.585,-37.109,179.181,5.432,149.196
C03203=1211.602,-119.834,-37.099,179.180,5.432,149.197
C03204=1211.608,-120.085,-37.090,179.177,5.432,149.197
C03205=1211.613,-120.334,-37.080,179.175,5.432,149.198
C03206=1211.618,-120.585,-37.071,179.173,5.431,149.198
C03207=1211.623,-120.834,-37.061,179.170,5.432,149.199
C03208=1211.629,-121.084,-37.051,179.168,5.431,149.200
C03209=1211.634,-121.333,-37.042,179.166,5.432,149.201
C03210=1211.639,-121.583,-37.033,179.164,5.431,149.201
C03211=1211.645,-121.833,-37.023,179.161,5.431,149.202
C03212=1211.650,-122.083,-37.014,179.159,5.432,149.203
C03213=1211.656,-122.333,-37.004,179.157,5.431,149.203
C03214=1211.661,-122.582,-36.995,179.155,5.431,149.204
C03215=1211.666,-122.832,-36.986,179.152,5.431,149.204
C03216=1211.671,-123.081,-36.976,179.150,5.431,149.205
C03217=1211.677,-123.331,-36.967,179.148,5.430,149.206
C03218=1211.682,-123.581,-36.958,179.146,5.431,149.206
C03219=1211.687,-123.831,-36.947,179.143,5.430,149.207
C03220=1211.692,-124.081,-36.938,179.142,5.430,149.208
C03221=1211.698,-124.331,-36.928,179.139,5.430,149.208
C03222=1211.703,-124.581,-36.919,179.137,5.430,149.209
C03223=1211.708,-124.830,-36.910,179.134,5.430,149.210
C03224=1211.713,-125.080,-36.900,179.133,5.430,149.210
C03225=1211.719,-125.330,-36.891,179.131,5.430,149.211
C03226=1211.724,-125.580,-36.882,179.128,5.430,149.212
C03227=1211.729,-125.829,-36.872,179.126,5.430,149.212
C03228=1211.735,-126.079,-36.863,179.124,5.429,149.213
C03229=1211.740,-126.329,-36.854,179.122,5.430,149.214
C03230=1211.745,-126.578,-36.844,179.119,5.429,149.214
C03231=1211.324,-126.589,-36.882,179.115,5.433,149.216
C03232=1211.319,-126.340,-36.892,179.118,5.433,149.215
C03233=1211.314,-126.090,-36.901,179.120,5.433,149.215
C03234=1211.308,-125.840,-36.910,179.122,5.433,149.214
C03235=1211.303,-125.590,-36.920,179.124,5.433,149.214
C03236=1211.298,-125.340,-36.929,179.127,5.433,149.213
C03237=1211.292,-125.090,-36.938,179.128,5.433,149.212
C03238=1211.287,-124.841,-36.948,179.130,5.433,149.212
C03239=1211.282,-124.591,-36.957,179.133,5.433,149.211
C03240=1211.276,-124.341,-36.966,179.135,5.433,149.210
C03241=1211.271,-124.092,-36.976,179.137,5.434,149.210
C03242=1211.265,-123.842,-36.985,179.139,5.433,149.209
C03243=1211.260,-123.592,-36.994,179.142,5.434,149.208
C03244=1211.255,-123.343,-37.004,179.144,5.434,149.208
C03245=1211.249,-123.092,-37.013,179.146,5.434,149.207
C03246=1211.244,-122.843,-37.023,179.148,5.434,149.206
C03247=1211.239,-122.593,-37.032,179.151,5.435,149.206
C03248=1211.233,-122.343,-37.041,179.153,5.434,149.205
C03249=1211.228,-122.094,-37.051,179.155,5.435,149.204
C03250=1211.223,-121.844,-37.060,179.157,5.435,149.204
C03251=1211.218,-121.595,-37.070,179.159,5.434,149.203
C03252=1211.213,-121.344,-37.079,179.162,5.435,149.202
C03253=1211.207,-121.094,-37.089,179.164,5.434,149.202
C03254=1211.202,-120.845,-37.098,179.166,5.435,149.201
C03255=1211.196,-120.594,-37.108,179.168,5.435,149.201
C03256=1211.192,-120.345,-37.117,179.171,5.435,149.200
C03257=1211.186,-120.095,-37.126,179.172,5.435,149.199
C03258=1211.181,-119.846,-37.137,179.175,5.436,149.199
C03259=1211.176,-119.596,-37.145,179.177,5.435,149.198
C03260=1211.170,-119.346,-37.156,179.180,5.436,149.197
C03261=1211.165,-119.097,-37.165,179.181,5.436,149.197
C03262=1211.160,-118.846,-37.175,179.184,5.436,149.196
C03263=1211.155,-118.596,-37.184,179.186,5.436,149.195
C03264=1211.149,-118.347,-37.194,179.189,5.436,149.195
C03265=1211.144,-118.097,-37.203,179.191,5.436,149.194
C03266=1211.139,-117.848,-37.213,179.193,5.436,149.193
C03267=1211.133,-117.598,-37.222,179.195,5.436,149.193
C03268=1211.128,-117.348,-37.232,179.197,5.436,149.192
C03269=1211.122,-117.098,-37.241,179.200,5.436,149.191
C03270=1211.118,-116.848,-37.251,179.202,5.436,149.191
C03271=1211.113,-116.599,-37.262,179.204,5.436,149.190
C03272=1211.107,-116.349,-37.270,179.206,5.436,149.190
C03273=1211.102,-116.099,-37.281,179.209,5.437,149.189
C03274=1211.097,-115.850,-37.290,179.211,5.436,149.188
C03275=1211.091,-115.600,-37.300,179.213,5.437,149.187
C03276=1211.086,-115.350,-37.309,179.215,5.437,149.187
C03277=1211.081,-115.100,-37.319,179.218,5.437,149.186
C03278=1211.075,-114.850,-37.329,179.220,5.437,149.185
C03279=1211.070,-114.601,-37.338,179.222,5.437,149.185
C03280=1211.065,-114.351,-37.349,179.224,5.437,149.184
C03281=1211.060,-114.102,-37.358,179.227,5.438,149.184
C03282=1211.054,-113.852,-37.368,179.229,5.437,149.183
C03283=1211.050,-113.602,-37.378,179.231,5.438,149.182
C03284=1211.044,-113.352,-37.387,179.233,5.438,149.182
C03285=1211.039,-113.102,-37.397,179.235,5.437,149.181
C03286=1211.033,-112.853,-37.407,179.238,5.438,149.180
C03287=1211.027,-112.603,-37.416,179.239,5.438,149.180
C03288=1211.023,-112.353,-37.426,179.242,5.438,149.179
C03289=1211.017,-112.103,-37.437,179.244,5.438,149.178
C03290=1211.012,-111.853,-37.446,179.247,5.438,149.178
C03291=1211.007,-111.604,-37.456,179.248,5.438,149.177
C03292=1211.002,-111.354,-37.465,179.251,5.439,149.176
C03293=1210.997,-111.104,-37.476,179.253,5.438,149.176
C03294=1210.991,-110.854,-37.485,179.256,5.439,149.175
C03295=1210.986,-110.605,-37.495,179.258,5.439,149.174
C03296=1210.980,-110.355,-37.505,179.260,5.439,149.174
C03297=1210.974,-110.105,-37.515,179.262,5.439,149.173
C03298=1210.970,-109.855,-37.525,179.265,5.439,149.172
C03299=1210.965,-109.606,-37.535,179.267,5.439,149.172
C03300=1210.960,-109.356,-37.545,179.269,5.439,149.171
C03301=1210.954,-109.106,-37.554,179.271,5.439,149.170
C03302=1210.949,-108.856,-37.565,179.274,5.439,149.170
C03303=1210.944,-108.607,-37.574,179.276,5.439,149.169
C03304=1210.938,-108.357,-37.584,179.278,5.440,149.169
C03305=1210.933,-108.108,-37.595,179.280,5.440,149.168
C03306=1210.928,-107.857,-37.604,179.283,5.440,149.167
C03307=1210.923,-107.608,-37.614,179.285,5.440,149.166
C03308=1210.917,-107.358,-37.624,179.287,5.440,149.166
C03309=1210.912,-107.109,-37.634,179.289,5.440,149.165
C03310=1210.907,-106.859,-37.645,179.292,5.440,149.164
C03311=1210.901,-106.608,-37.654,179.294,5.440,149.164
C03312=1210.896,-106.359,-37.664,179.296,5.441,149.163
C03313=1210.891,-106.109,-37.674,179.298,5.440,149.163
C03314=1210.886,-105.859,-37.684,179.301,5.441,149.162
C03315=1210.880,-105.610,-37.695,179.303,5.440,149.161
C03316=1210.875,-105.361,-37.704,179.306,5.441,149.160
C03317=1210.870,-105.110,-37.714,179.308,5.441,149.160
C03318=1210.864,-104.860,-37.724,179.310,5.441,149.159
C03319=1210.860,-104.611,-37.734,179.312,5.441,149.158
C03320=1210.855,-104.361,-37.744,179.315,5.441,149.158
C03321=1210.849,-104.111,-37.755,179.317,5.441,149.157
C03322=1210.843,-103.862,-37.765,179.319,5.442,149.157
C03323=1210.839,-103.612,-37.775,179.321,5.441,149.156
C03324=1210.834,-103.362,-37.785,179.324,5.442,149.155
C03325=1210.828,-103.113,-37.795,179.326,5.441,149.154
C03326=1210.822,-102.863,-37.805,179.328,5.442,149.154
C03327=1210.818,-102.613,-37.815,179.330,5.442,149.153
C03328=1210.812,-102.363,-37.825,179.333,5.442,149.153
C03329=1210.807,-102.113,-37.835,179.335,5.442,149.152
C03330=1210.802,-101.863,-37.846,179.337,5.443,149.151
C03331=1210.797,-101.614,-37.855,179.339,5.442,149.151
C03332=1210.791,-101.342,-37.867,179.342,5.443,149.150
C03333=1210.786,-101.071,-37.878,179.344,5.442,149.149
C03334=1210.779,-100.800,-37.889,179.347,5.443,149.148
C03335=1210.774,-100.529,-37.900,179.350,5.443,149.148
C03336=1210.768,-100.279,-37.910,179.352,5.443,149.147
C03337=1210.763,-100.029,-37.921,179.354,5.443,149.146
C03338=1210.758,-99.780,-37.931,179.356,5.443,149.146
C03339=1210.753,-99.530,-37.941,179.359,5.443,149.145
C03340=1210.748,-99.280,-37.951,179.361,5.443,149.144
C03341=1210.742,-99.031,-37.961,179.363,5.444,149.144
C03342=1210.737,-98.780,-37.972,179.365,5.443,149.143
C03343=1210.732,-98.531,-37.982,179.368,5.444,149.142
C03344=1210.726,-98.281,-37.992,179.370,5.444,149.142
C03345=1210.722,-98.031,-38.002,179.372,5.444,149.141
C03346=1210.716,-97.782,-38.013,179.374,5.444,149.140
C03347=1210.711,-97.533,-38.023,179.377,5.444,149.140
C03348=1210.706,-97.283,-38.034,179.379,5.444,149.139
C03349=1210.700,-97.033,-38.044,179.381,5.445,149.138
C03350=1210.695,-96.783,-38.055,179.384,5.444,149.138
C03351=1210.690,-96.533,-38.065,179.386,5.445,149.137
C03352=1210.684,-96.284,-38.075,179.388,5.444,149.136
C03353=1210.680,-96.034,-38.085,179.391,5.445,149.136
C03354=1210.674,-95.784,-38.095,179.393,5.445,149.135
C03355=1210.669,-95.534,-38.106,179.395,5.445,149.134
C03356=1210.664,-95.284,-38.116,179.397,5.445,149.134
C03357=1210.659,-95.035,-38.127,179.400,5.445,149.133
C03358=1210.653,-94.785,-38.138,179.402,5.445,149.132
C03359=1210.648,-94.536,-38.148,179.405,5.445,149.132
C03360=1210.643,-94.285,-38.158,179.406,5.445,149.131
C03361=1210.637,-94.036,-38.169,179.409,5.446,149.130
C03362=1210.632,-93.786,-38.179,179.411,5.445,149.130
C03363=1210.627,-93.537,-38.190,179.414,5.446,149.129
C03364=1210.622,-93.286,-38.201,179.416,5.445,149.128
C03365=1210.616,-93.037,-38.211,179.418,5.446,149.128
C03366=1210.611,-92.787,-38.221,179.420,5.446,149.127
C03367=1210.606,-92.537,-38.232,179.423,5.446,149.126
C03368=1210.600,-92.288,-38.243,179.426,5.447,149.126
C03369=1210.596,-92.038,-38.253,179.428,5.446,149.125
C03370=1210.591,-91.789,-38.263,179.430,5.447,149.124
C03371=1210.586,-91.539,-38.273,179.432,5.447,149.124
C03372=1210.580,-91.289,-38.284,179.435,5.447,149.123
C03373=1210.575,-91.039,-38.295,179.437,5.447,149.122
C03374=1210.570,-90.790,-38.305,179.439,5.447,149.122
C03375=1210.565,-90.540,-38.316,179.441,5.447,149.121
C03376=1210.559,-90.291,-38.327,179.444,5.448,149.120
C03377=1210.554,-90.040,-38.337,179.446,5.447,149.120
C03378=1210.549,-89.791,-38.347,179.448,5.448,149.119
C03379=1210.544,-89.541,-38.358,179.450,5.447,149.118
C03380=1210.539,-89.292,-38.369,179.453,5.448,149.118
C03381=1210.533,-89.041,-38.380,179.455,5.448,149.117
C03382=1210.527,-88.792,-38.390,179.457,5.448,149.116
C03383=1210.522,-88.542,-38.402,179.459,5.448,149.116
C03384=1210.517,-88.292,-38.412,179.462,5.448,149.115
C03385=1210.512,-88.042,-38.422,179.464,5.448,149.114
C03386=1210.507,-87.793,-38.433,179.467,5.448,149.114
C03387=1210.502,-87.543,-38.444,179.469,5.449,149.113
C03388=1210.496,-87.293,-38.454,179.471,5.449,149.112
C03389=1210.491,-87.044,-38.465,179.474,5.449,149.112
C03390=1210.486,-86.794,-38.476,179.476,5.449,149.111
C03391=1210.481,-86.544,-38.486,179.479,5.449,149.110
C03392=1210.475,-86.295,-38.497,179.481,5.449,149.109
C03393=1210.470,-86.045,-38.508,179.483,5.450,149.109
C03394=1210.465,-85.795,-38.518,179.485,5.449,149.108
C03395=1210.460,-85.546,-38.529,179.488,5.450,149.108
C03396=1210.454,-85.295,-38.540,179.490,5.449,149.107
C03397=1210.449,-85.046,-38.551,179.492,5.450,149.106
C03398=1210.444,-84.796,-38.562,179.494,5.449,149.105
C03399=1210.439,-84.547,-38.573,179.497,5.450,149.105
C03400=1210.434,-84.297,-38.583,179.499,5.451,149.104
C03401=1210.428,-84.047,-38.594,179.501,5.450,149.104
C03402=1210.424,-83.798,-38.605,179.504,5.451,149.103
C03403=1210.419,-83.547,-38.615,179.506,5.450,149.102
C03404=1210.413,-83.298,-38.626,179.509,5.451,149.101
C03405=1210.407,-83.048,-38.637,179.510,5.451,149.101
C03406=1210.402,-82.799,-38.648,179.513,5.451,149.100
C03407=1210.397,-82.549,-38.659,179.515,5.451,149.100
C03408=1210.393,-82.299,-38.670,179.518,5.451,149.099
C03409=1210.387,-82.050,-38.680,179.520,5.451,149.098
C03410=1210.382,-81.800,-38.692,179.523,5.451,149.097
C03411=1210.376,-81.550,-38.703,179.525,5.452,149.097
C03412=1210.371,-81.300,-38.714,179.527,5.452,149.096
C03413=1210.366,-81.050,-38.724,179.530,5.452,149.095
C03414=1210.361,-80.801,-38.735,179.532,5.452,149.095
C03415=1210.356,-80.551,-38.746,179.534,5.452,149.094
C03416=1210.350,-80.302,-38.757,179.536,5.452,149.093
C03417=1210.345,-80.052,-38.768,179.539,5.452,149.093
C03418=1210.340,-79.802,-38.779,179.541,5.453,149.092
C03419=1210.335,-79.553,-38.790,179.543,5.453,149.091
C03420=1210.330,-79.303,-38.801,179.546,5.453,149.091
C03421=1210.324,-79.053,-38.813,179.548,5.453,149.090
C03422=1210.319,-78.803,-38.823,179.551,5.453,149.089
C03423=1210.314,-78.554,-38.834,179.553,5.453,149.089
C03424=1210.309,-78.303,-38.845,179.556,5.454,149.088
C03425=1210.303,-78.054,-38.856,179.557,5.454,149.087
C03426=1210.298,-77.805,-38.868,179.560,5.454,149.087
C03427=1210.293,-77.554,-38.878,179.562,5.454,149.086
C03428=1210.288,-77.305,-38.889,179.565,5.454,149.085
C03429=1210.283,-77.055,-38.901,179.567,5.455,149.085
C03430=1210.277,-76.806,-38.911,179.569,5.454,149.084
C03431=1210.272,-76.556,-38.922,179.572,5.455,149.083
C03432=1210.267,-76.306,-38.934,179.574,5.455,149.083
C03433=1210.261,-76.057,-38.945,179.576,5.455,149.082
C03434=1210.257,-75.807,-38.956,179.578,5.455,149.081
C03435=1210.251,-75.557,-38.967,179.581,5.455,149.081
C03436=1210.246,-75.287,-38.979,179.584,5.456,149.080
C03437=1210.240,-75.016,-38.991,179.586,5.455,149.079
C03438=1210.235,-74.745,-39.004,179.588,5.456,149.078
C03439=1210.228,-74.475,-39.015,179.591,5.456,149.078
C03440=1210.224,-74.225,-39.027,179.593,5.456,149.077
C03441=1210.219,-73.975,-39.037,179.596,5.456,149.076
C03442=1210.213,-73.726,-39.049,179.598,5.456,149.076
C03443=1210.208,-73.476,-39.060,179.601,5.456,149.075
C03444=1210.203,-73.227,-39.071,179.603,5.457,149.074
C03445=1210.198,-72.976,-39.083,179.605,5.457,149.074
C03446=1210.192,-72.727,-39.093,179.608,5.457,149.073
C03447=1210.187,-72.477,-39.105,179.610,5.457,149.072
C03448=1210.182,-72.228,-39.117,179.612,5.457,149.072
C03449=1210.177,-71.978,-39.127,179.615,5.458,149.071
C03450=1210.171,-71.728,-39.139,179.617,5.457,149.070
C03451=1210.166,-71.479,-39.150,179.620,5.458,149.069
C03452=1210.162,-71.229,-39.161,179.622,5.457,149.069
C03453=1210.155,-70.979,-39.172,179.624,5.458,149.068
C03454=1210.151,-70.729,-39.183,179.626,5.458,149.068
C03455=1210.145,-70.480,-39.195,179.629,5.458,149.067
C03456=1210.141,-70.230,-39.207,179.631,5.459,149.066
C03457=1210.135,-69.981,-39.218,179.634,5.458,149.065
C03458=1210.130,-69.731,-39.229,179.636,5.459,149.065
C03459=1210.125,-69.481,-39.240,179.638,5.458,149.064
C03460=1210.119,-69.231,-39.252,179.640,5.459,149.064
C03461=1210.114,-68.982,-39.263,179.643,5.459,149.063
C03462=1210.109,-68.732,-39.275,179.645,5.459,149.062
C03463=1210.104,-68.482,-39.286,179.648,5.460,149.061
C03464=1210.099,-68.232,-39.298,179.650,5.459,149.061
C03465=1210.094,-67.983,-39.309,179.653,5.460,149.060
C03466=1210.089,-67.734,-39.320,179.655,5.460,149.059
C03467=1210.083,-67.483,-39.331,179.657,5.460,149.059
C03468=1210.078,-67.234,-39.343,179.660,5.461,149.058
C03469=1210.073,-66.984,-39.354,179.662,5.460,149.057
C03470=1210.068,-66.734,-39.366,179.664,5.461,149.057
C03471=1210.062,-66.485,-39.377,179.666,5.461,149.056
C03472=1210.057,-66.235,-39.389,179.669,5.461,149.055
C03473=1210.052,-65.985,-39.400,179.672,5.461,149.055
C03474=1210.047,-65.736,-39.412,179.674,5.461,149.054
C03475=1210.042,-65.486,-39.424,179.677,5.462,149.053
C03476=1210.036,-65.237,-39.434,179.678,5.462,149.053
C03477=1210.031,-64.987,-39.446,179.681,5.462,149.052
C03478=1210.026,-64.737,-39.458,179.683,5.462,149.051
C03479=1210.021,-64.487,-39.470,179.686,5.462,149.051
C03480=1210.016,-64.238,-39.481,179.688,5.463,149.050
C03481=1210.011,-63.988,-39.493,179.690,5.462,149.049
C03482=1210.005,-63.739,-39.504,179.693,5.463,149.048
C03483=1210.000,-63.489,-39.516,179.696,5.463,149.048
C03484=1209.995,-63.239,-39.527,179.697,5.463,149.047
C03485=1209.990,-62.989,-39.539,179.700,5.464,149.047
C03486=1209.985,-62.739,-39.551,179.702,5.463,149.046
C03487=1209.980,-62.490,-39.562,179.705,5.464,149.045
C03488=1209.974,-62.240,-39.574,179.707,5.464,149.044
C03489=1209.969,-61.991,-39.585,179.709,5.464,149.044
C03490=1209.964,-61.741,-39.597,179.712,5.464,149.043
C03491=1209.958,-61.491,-39.608,179.714,5.464,149.042
C03492=1209.954,-61.241,-39.620,179.716,5.465,149.042
C03493=1209.948,-60.991,-39.632,179.719,5.465,149.041
C03494=1209.944,-60.742,-39.644,179.721,5.465,149.040
C03495=1209.938,-60.493,-39.656,179.724,5.465,149.040
C03496=1209.933,-60.243,-39.667,179.726,5.465,149.039
C03497=1209.928,-59.993,-39.679,179.729,5.465,149.038
C03498=1209.922,-59.744,-39.690,179.731,5.466,149.038
C03499=1209.917,-59.494,-39.702,179.733,5.465,149.037
C03500=1209.912,-59.244,-39.713,179.736,5.466,149.036
C03501=1209.907,-58.994,-39.725,179.738,5.466,149.036
C03502=1209.902,-58.745,-39.737,179.740,5.466,149.035
C03503=1209.897,-58.495,-39.749,179.743,5.467,149.034
C03504=1209.891,-58.245,-39.761,179.745,5.467,149.034
C03505=1209.887,-57.996,-39.772,179.748,5.467,149.033
C03506=1209.881,-57.746,-39.784,179.750,5.467,149.032
C03507=1209.876,-57.496,-39.796,179.752,5.467,149.032
C03508=1209.871,-57.247,-39.808,179.755,5.468,149.031
C03509=1209.866,-56.997,-39.820,179.757,5.468,149.030
C03510=1209.861,-56.747,-39.832,179.759,5.468,149.030
C03511=1209.856,-56.497,-39.843,179.762,5.468,149.029
C03512=1209.850,-56.249,-39.855,179.764,5.468,149.028
C03513=1209.845,-55.999,-39.867,179.767,5.469,149.028
C03514=1209.840,-55.749,-39.879,179.769,5.469,149.027
C03515=1209.835,-55.499,-39.890,179.771,5.469,149.026
C03516=1209.829,-55.250,-39.903,179.774,5.469,149.025
C03517=1209.825,-55.000,-39.914,179.776,5.469,149.025
C03518=1209.819,-54.750,-39.926,179.778,5.470,149.024
C03519=1209.814,-54.500,-39.938,179.781,5.470,149.024
C03520=1209.809,-54.251,-39.951,179.783,5.470,149.023
C03521=1209.804,-54.001,-39.962,179.786,5.470,149.022
C03522=1209.799,-53.752,-39.974,179.788,5.471,149.021
C03523=1209.794,-53.502,-39.987,179.791,5.470,149.021
C03524=1209.788,-53.252,-39.998,179.793,5.471,149.020
C03525=1209.783,-53.003,-40.010,179.795,5.470,149.019
C03526=1209.778,-52.753,-40.022,179.798,5.471,149.019
C03527=1209.773,-52.503,-40.034,179.800,5.472,149.018
C03528=1209.767,-52.253,-40.046,179.802,5.471,149.017
C03529=1209.763,-52.004,-40.058,179.805,5.472,149.017
C03530=1209.758,-51.755,-40.070,179.808,5.472,149.016
C03531=1209.752,-51.505,-40.082,179.810,5.472,149.015
C03532=1209.747,-51.255,-40.094,179.812,5.472,149.015
C03533=1209.742,-51.005,-40.106,179.815,5.473,149.014
C03534=1209.737,-50.756,-40.118,179.817,5.473,149.013
C03535=1209.732,-50.506,-40.130,179.820,5.473,149.013
C03536=1209.726,-50.256,-40.142,179.822,5.473,149.012
C03537=1209.721,-50.007,-40.155,179.824,5.473,149.011
C03538=1209.716,-49.757,-40.167,179.827,5.474,149.011
C03539=1209.710,-49.507,-40.178,179.829,5.474,149.010
C03540=1209.705,-49.238,-40.192,179.831,5.474,149.009
C03541=1209.700,-48.967,-40.205,179.834,5.475,149.009
C03542=1209.694,-48.698,-40.218,179.837,5.475,149.008
C03543=1209.689,-48.427,-40.231,179.839,5.474,149.007
C03544=1209.684,-48.178,-40.243,179.842,5.475,149.006
C03545=1209.678,-47.928,-40.255,179.845,5.475,149.005
C03546=1209.673,-47.679,-40.268,179.846,5.475,149.005
C03547=1209.668,-47.429,-40.280,179.849,5.476,149.004
C03548=1209.663,-47.179,-40.292,179.852,5.476,149.004
C03549=1209.658,-46.930,-40.304,179.854,5.476,149.003
C03550=1209.653,-46.680,-40.316,179.856,5.476,149.002
C03551=1209.648,-46.430,-40.328,179.859,5.477,149.002
C03552=1209.643,-46.180,-40.341,179.861,5.476,149.001
C03553=1209.637,-45.931,-40.353,179.864,5.477,149.000
C03554=1209.632,-45.681,-40.365,179.866,5.477,148.999
C03555=1209.627,-45.431,-40.377,179.868,5.477,148.999
C03556=1209.622,-45.182,-40.390,179.871,5.478,148.998
C03557=1209.617,-44.933,-40.403,179.873,5.478,148.998
C03558=1209.611,-44.683,-40.414,179.875,5.478,148.997
C03559=1209.606,-44.433,-40.427,179.878,5.478,148.996
C03560=1209.601,-44.183,-40.439,179.881,5.479,148.995
C03561=1209.596,-43.933,-40.452,179.883,5.479,148.995
C03562=1209.591,-43.683,-40.464,179.885,5.479,148.994
C03563=1209.586,-43.434,-40.476,179.888,5.479,148.993
C03564=1209.581,-43.185,-40.488,179.890,5.479,148.993
C03565=1209.576,-42.935,-40.500,179.892,5.480,148.992
C03566=1209.571,-42.686,-40.513,179.895,5.480,148.991
C03567=1209.565,-42.436,-40.525,179.897,5.480,148.991
C03568=1209.561,-42.186,-40.538,179.900,5.481,148.990
C03569=1209.556,-41.937,-40.550,179.902,5.481,148.989
C03570=1209.550,-41.687,-40.562,179.905,5.481,148.989
C03571=1209.545,-41.437,-40.575,179.907,5.481,148.988
C03572=1209.540,-41.188,-40.587,179.910,5.482,148.987
C03573=1209.534,-40.938,-40.599,179.912,5.481,148.987
C03574=1209.529,-40.689,-40.612,179.915,5.482,148.986
C03575=1209.525,-40.439,-40.625,179.917,5.483,148.985
C03576=1209.519,-40.189,-40.637,179.919,5.482,148.985
C03577=1209.514,-39.939,-40.650,179.922,5.483,148.984
C03578=1209.508,-39.690,-40.663,179.924,5.483,148.983
C03579=1209.503,-39.441,-40.675,179.926,5.483,148.983
C03580=1209.498,-39.190,-40.687,179.929,5.483,148.982
C03581=1209.493,-38.941,-40.700,179.932,5.484,148.981
C03582=1209.488,-38.691,-40.713,179.934,5.483,148.980
C03583=1209.483,-38.442,-40.725,179.936,5.484,148.980
C03584=1209.478,-38.192,-40.737,179.939,5.484,148.979
C03585=1209.473,-37.943,-40.750,179.941,5.484,148.979
C03586=1209.468,-37.693,-40.763,179.943,5.485,148.978
C03587=1209.463,-37.443,-40.775,179.946,5.485,148.977
C03588=1209.457,-37.193,-40.787,179.948,5.485,148.976
C03589=1209.452,-36.944,-40.800,179.951,5.486,148.976
C03590=1209.447,-36.694,-40.813,179.953,5.486,148.975
C03591=1209.442,-36.445,-40.826,179.956,5.486,148.974
C03592=1209.437,-36.195,-40.839,179.958,5.486,148.974
C03593=1209.431,-35.945,-40.850,179.961,5.487,148.973
C03594=1209.426,-35.696,-40.863,179.963,5.487,148.972
C03595=1209.422,-35.446,-40.876,179.965,5.487,148.972
C03596=1209.417,-35.197,-40.889,179.968,5.488,148.971
C03597=1209.412,-34.947,-40.901,179.970,5.488,148.970
C03598=1209.406,-34.698,-40.914,179.972,5.488,148.970
C03599=1209.401,-34.447,-40.927,179.975,5.488,148.969
C03600=1209.396,-34.198,-40.939,179.978,5.489,148.968
C03601=1209.391,-33.948,-40.952,179.980,5.488,148.968
C03602=1209.385,-33.699,-40.964,179.982,5.489,148.967
C03603=1209.381,-33.449,-40.977,179.985,5.489,148.966
C03604=1209.375,-33.199,-40.991,179.988,5.490,148.966
C03605=1209.370,-32.950,-41.003,179.989,5.490,148.965
C03606=1209.365,-32.700,-41.016,179.992,5.490,148.964
C03607=1209.360,-32.451,-41.029,179.995,5.491,148.964
C03608=1209.355,-32.201,-41.041,179.997,5.490,148.963
C03609=1209.349,-31.952,-41.055,179.999,5.491,148.962
C03610=1209.344,-31.701,-41.067,-179.998,5.491,148.962
C03611=1209.339,-31.452,-41.079,-179.996,5.491,148.961
C03612=1209.334,-31.203,-41.092,-179.993,5.492,148.960
C03613=1209.329,-30.952,-41.106,-179.990,5.492,148.959
C03614=1209.324,-30.703,-41.118,-179.988,5.492,148.959
C03615=1209.319,-30.454,-41.131,-179.986,5.492,148.958
C03616=1209.314,-30.204,-41.143,-179.984,5.493,148.958
C03617=1209.309,-29.954,-41.156,-179.981,5.493,148.957
C03618=1209.303,-29.705,-41.170,-179.979,5.493,148.956
C03619=1209.298,-29.455,-41.182,-179.976,5.494,148.956
C03620=1209.294,-29.205,-41.195,-179.973,5.494,148.955
C03621=1209.288,-28.956,-41.208,-179.971,5.495,148.954
C03622=1209.283,-28.706,-41.221,-179.969,5.494,148.953
C03623=1209.278,-28.457,-41.235,-179.966,5.495,148.953
C03624=1209.273,-28.208,-41.247,-179.963,5.495,148.952
C03625=1209.267,-27.958,-41.260,-179.961,5.495,148.951
C03626=1209.263,-27.708,-41.273,-179.959,5.496,148.951
C03627=1209.258,-27.459,-41.286,-179.957,5.496,148.950
C03628=1209.252,-27.208,-41.300,-179.954,5.497,148.949
C03629=1209.247,-26.959,-41.312,-179.952,5.496,148.949
C03630=1209.242,-26.710,-41.325,-179.949,5.497,148.948
C03631=1209.238,-26.460,-41.338,-179.946,5.497,148.947
C03632=1209.232,-26.210,-41.351,-179.944,5.498,148.947
C03633=1209.227,-25.961,-41.363,-179.942,5.497,148.946
C03634=1209.223,-25.711,-41.377,-179.939,5.498,148.945
C03635=1209.217,-25.462,-41.390,-179.936,5.498,148.945
C03636=1209.212,-25.212,-41.403,-179.935,5.498,148.944
C03637=1209.206,-24.962,-41.417,-179.932,5.499,148.943
C03638=1209.201,-24.713,-41.429,-179.929,5.499,148.943
C03639=1209.197,-24.463,-41.442,-179.927,5.500,148.942
C03640=1209.191,-24.214,-41.456,-179.925,5.500,148.941
C03641=1209.187,-23.964,-41.469,-179.922,5.500,148.941
C03642=1209.181,-23.714,-41.482,-179.919,5.501,148.940
C03643=1209.176,-23.465,-41.495,-179.917,5.501,148.939
C03644=1209.171,-23.195,-41.508,-179.915,5.501,148.939
C03645=1209.165,-22.926,-41.523,-179.912,5.501,148.938
